ABB RAPID module: P36.mod

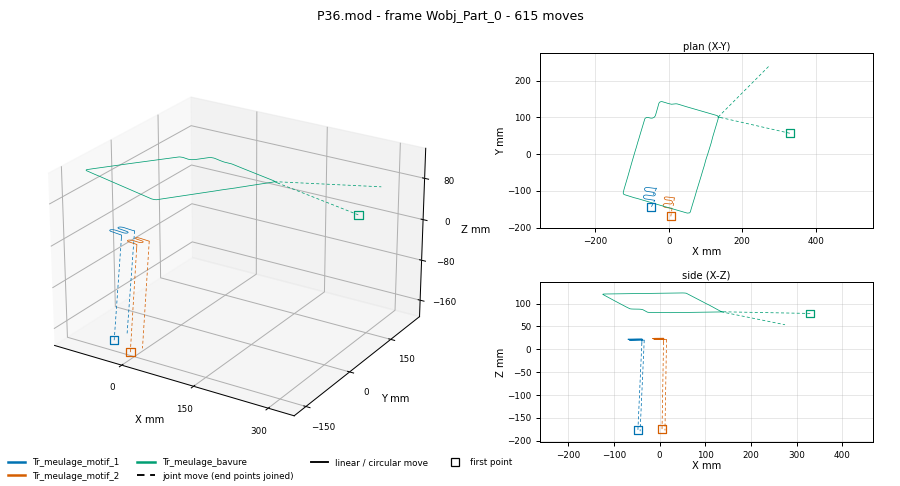
[picture p0: tool path of P36.mod in frame Wobj_Part_0, 615 of 623 moves have a stored position in this frame; points joined in program order, loops and branches not executed]
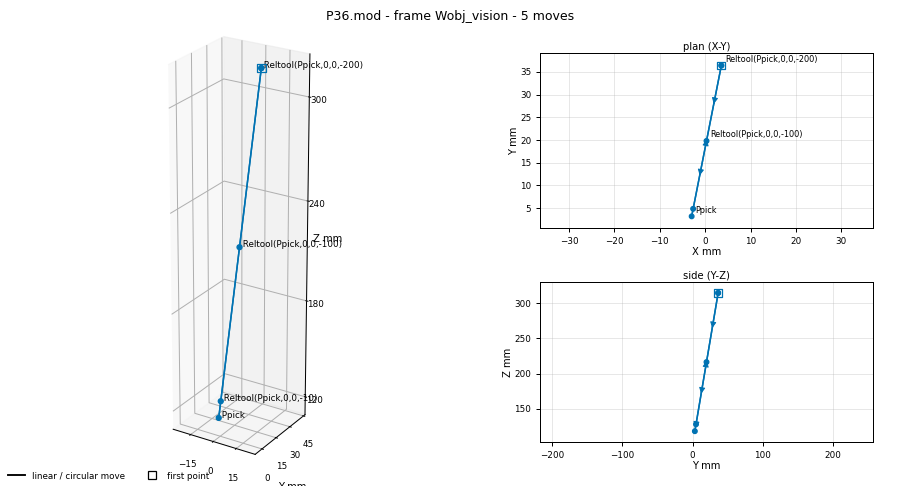
[picture p1: tool path of P36.mod in frame Wobj_vision, 5 of 623 moves have a stored position in this frame; points joined in program order, loops and branches not executed]
MODULE P36
	LOCAL CONST Speeddata vitesse_Tronconnage :=[10, 500, 0, 0];
	LOCAL CONST Robtarget Tr_meulage_motif_1_App1 :=[[-47.3344757449952,-143.415724704918,-176.118398279714],[-0.000994403231452177,0.0225685468013881,0.0440075228376034,0.998775755508305],[0,0,0,0],[8.999999E+09,8.999999E+09,8.999999E+09,8.999999E+09,8.999999E+09,8.999999E+09]];
	LOCAL CONST Robtarget Tr_meulage_motif_1_App2 :=[[-38.7855564044373,-126.704810844621,12.9521211992956],[-0.000994403231452177,0.0225685468013881,0.0440075228376034,0.998775755508305],[0,0,0,0],[8.999999E+09,8.999999E+09,8.999999E+09,8.999999E+09,8.999999E+09,8.999999E+09]];
	LOCAL CONST Robtarget Tr_meulage_motif_1_P0 :=[[-38.33561328125,-125.8252890625,22.903201171875],[-0.000994403231452177,0.0225685468013881,0.0440075228376034,0.998775755508305],[0,0,0,0],[8.999999E+09,8.999999E+09,8.999999E+09,8.999999E+09,8.999999E+09,8.999999E+09]];
	LOCAL CONST Robtarget Tr_meulage_motif_1_P1 :=[[-39.3248359375,-125.679359375,22.8911484375],[-0.000994403231452177,0.0225685468013881,0.0440075228376034,0.998775755508305],[0,0,0,0],[8.999999E+09,8.999999E+09,8.999999E+09,8.999999E+09,8.999999E+09,8.999999E+09]];
	LOCAL CONST Robtarget Tr_meulage_motif_1_P2 :=[[-40.3140546875,-125.533421875,22.879095703125],[-0.000994403231452177,0.0225685468013881,0.0440075228376034,0.998775755508305],[0,0,0,0],[8.999999E+09,8.999999E+09,8.999999E+09,8.999999E+09,8.999999E+09,8.999999E+09]];
	LOCAL CONST Robtarget Tr_meulage_motif_1_P3 :=[[-41.30327734375,-125.3874921875,22.867041015625],[-0.000994403231452177,0.0225685468013881,0.0440075228376034,0.998775755508305],[0,0,0,0],[8.999999E+09,8.999999E+09,8.999999E+09,8.999999E+09,8.999999E+09,8.999999E+09]];
	LOCAL CONST Robtarget Tr_meulage_motif_1_P4 :=[[-42.29249609375,-125.2415546875,22.85498828125],[-0.000994403231452177,0.0225685468013881,0.0440075228376034,0.998775755508305],[0,0,0,0],[8.999999E+09,8.999999E+09,8.999999E+09,8.999999E+09,8.999999E+09,8.999999E+09]];
	LOCAL CONST Robtarget Tr_meulage_motif_1_P5 :=[[-43.28171875,-125.095625,22.842935546875],[-0.000994403231452177,0.0225685468013881,0.0440075228376034,0.998775755508305],[0,0,0,0],[8.999999E+09,8.999999E+09,8.999999E+09,8.999999E+09,8.999999E+09,8.999999E+09]];
	LOCAL CONST Robtarget Tr_meulage_motif_1_P6 :=[[-44.2709375,-124.9496953125,22.8308828125],[-0.000994403231452177,0.0225685468013881,0.0440075228376034,0.998775755508305],[0,0,0,0],[8.999999E+09,8.999999E+09,8.999999E+09,8.999999E+09,8.999999E+09,8.999999E+09]];
	LOCAL CONST Robtarget Tr_meulage_motif_1_P7 :=[[-45.26016015625,-124.8037578125,22.818828125],[-0.000994403231452177,0.0225685468013881,0.0440075228376034,0.998775755508305],[0,0,0,0],[8.999999E+09,8.999999E+09,8.999999E+09,8.999999E+09,8.999999E+09,8.999999E+09]];
	LOCAL CONST Robtarget Tr_meulage_motif_1_P8 :=[[-46.2493828125,-124.657828125,22.806775390625],[-0.000994403231452177,0.0225685468013881,0.0440075228376034,0.998775755508305],[0,0,0,0],[8.999999E+09,8.999999E+09,8.999999E+09,8.999999E+09,8.999999E+09,8.999999E+09]];
	LOCAL CONST Robtarget Tr_meulage_motif_1_P9 :=[[-47.2386015625,-124.511890625,22.79472265625],[-0.000994403231452177,0.0225685468013881,0.0440075228376034,0.998775755508305],[0,0,0,0],[8.999999E+09,8.999999E+09,8.999999E+09,8.999999E+09,8.999999E+09,8.999999E+09]];
	LOCAL CONST Robtarget Tr_meulage_motif_1_P10 :=[[-48.22782421875,-124.3659609375,22.782669921875],[-0.000994403231452177,0.0225685468013881,0.0440075228376034,0.998775755508305],[0,0,0,0],[8.999999E+09,8.999999E+09,8.999999E+09,8.999999E+09,8.999999E+09,8.999999E+09]];
	LOCAL CONST Robtarget Tr_meulage_motif_1_P11 :=[[-49.21704296875,-124.2200234375,22.770615234375],[-0.000994403231452177,0.0225685468013881,0.0440075228376034,0.998775755508305],[0,0,0,0],[8.999999E+09,8.999999E+09,8.999999E+09,8.999999E+09,8.999999E+09,8.999999E+09]];
	LOCAL CONST Robtarget Tr_meulage_motif_1_P12 :=[[-50.206265625,-124.07409375,22.7585625],[-0.000994403231452177,0.0225685468013881,0.0440075228376034,0.998775755508305],[0,0,0,0],[8.999999E+09,8.999999E+09,8.999999E+09,8.999999E+09,8.999999E+09,8.999999E+09]];
	LOCAL CONST Robtarget Tr_meulage_motif_1_P13 :=[[-51.195484375,-123.92815625,22.746509765625],[-0.000994403231452177,0.0225685468013881,0.0440075228376034,0.998775755508305],[0,0,0,0],[8.999999E+09,8.999999E+09,8.999999E+09,8.999999E+09,8.999999E+09,8.999999E+09]];
	LOCAL CONST Robtarget Tr_meulage_motif_1_P14 :=[[-52.18470703125,-123.7822265625,22.734455078125],[-0.000994403231452177,0.0225685468013881,0.0440075228376034,0.998775755508305],[0,0,0,0],[8.999999E+09,8.999999E+09,8.999999E+09,8.999999E+09,8.999999E+09,8.999999E+09]];
	LOCAL CONST Robtarget Tr_meulage_motif_1_P15 :=[[-53.1739296875,-123.6362890625,22.72240234375],[-0.000994403231452177,0.0225685468013881,0.0440075228376034,0.998775755508305],[0,0,0,0],[8.999999E+09,8.999999E+09,8.999999E+09,8.999999E+09,8.999999E+09,8.999999E+09]];
	LOCAL CONST Robtarget Tr_meulage_motif_1_P16 :=[[-54.1631484375,-123.490359375,22.710349609375],[-0.000994403231452177,0.0225685468013881,0.0440075228376034,0.998775755508305],[0,0,0,0],[8.999999E+09,8.999999E+09,8.999999E+09,8.999999E+09,8.999999E+09,8.999999E+09]];
	LOCAL CONST Robtarget Tr_meulage_motif_1_P17 :=[[-55.15237109375,-123.344421875,22.698296875],[-0.000994403231452177,0.0225685468013881,0.0440075228376034,0.998775755508305],[0,0,0,0],[8.999999E+09,8.999999E+09,8.999999E+09,8.999999E+09,8.999999E+09,8.999999E+09]];
	LOCAL CONST Robtarget Tr_meulage_motif_1_P18 :=[[-56.14158984375,-123.1984921875,22.6862421875],[-0.000994403231452177,0.0225685468013881,0.0440075228376034,0.998775755508305],[0,0,0,0],[8.999999E+09,8.999999E+09,8.999999E+09,8.999999E+09,8.999999E+09,8.999999E+09]];
	LOCAL CONST Robtarget Tr_meulage_motif_1_P19 :=[[-57.1308125,-123.0525546875,22.674189453125],[-0.000994403231452177,0.0225685468013881,0.0440075228376034,0.998775755508305],[0,0,0,0],[8.999999E+09,8.999999E+09,8.999999E+09,8.999999E+09,8.999999E+09,8.999999E+09]];
	LOCAL CONST Robtarget Tr_meulage_motif_1_P20 :=[[-58.12003125,-122.906625,22.66213671875],[-0.000994403231452177,0.0225685468013881,0.0440075228376034,0.998775755508305],[0,0,0,0],[8.999999E+09,8.999999E+09,8.999999E+09,8.999999E+09,8.999999E+09,8.999999E+09]];
	LOCAL CONST Robtarget Tr_meulage_motif_1_P21 :=[[-59.10925390625,-122.7606875,22.650083984375],[-0.000994403231452177,0.0225685468013881,0.0440075228376034,0.998775755508305],[0,0,0,0],[8.999999E+09,8.999999E+09,8.999999E+09,8.999999E+09,8.999999E+09,8.999999E+09]];
	LOCAL CONST Robtarget Tr_meulage_motif_1_P22 :=[[-60.0984765625,-122.6147578125,22.638029296875],[-0.000994403231452177,0.0225685468013881,0.0440075228376034,0.998775755508305],[0,0,0,0],[8.999999E+09,8.999999E+09,8.999999E+09,8.999999E+09,8.999999E+09,8.999999E+09]];
	LOCAL CONST Robtarget Tr_meulage_motif_1_P23 :=[[-61.0876953125,-122.4688203125,22.6259765625],[-0.000994403231452177,0.0225685468013881,0.0440075228376034,0.998775755508305],[0,0,0,0],[8.999999E+09,8.999999E+09,8.999999E+09,8.999999E+09,8.999999E+09,8.999999E+09]];
	LOCAL CONST Robtarget Tr_meulage_motif_1_P24 :=[[-62.07691796875,-122.322890625,22.613923828125],[-0.000994403231452177,0.0225685468013881,0.0440075228376034,0.998775755508305],[0,0,0,0],[8.999999E+09,8.999999E+09,8.999999E+09,8.999999E+09,8.999999E+09,8.999999E+09]];
	LOCAL CONST Robtarget Tr_meulage_motif_1_P25 :=[[-63.06613671875,-122.176953125,22.601869140625],[-0.000994403231452177,0.0225685468013881,0.0440075228376034,0.998775755508305],[0,0,0,0],[8.999999E+09,8.999999E+09,8.999999E+09,8.999999E+09,8.999999E+09,8.999999E+09]];
	LOCAL CONST Robtarget Tr_meulage_motif_1_P26 :=[[-64.03180859375,-121.92315625,22.57997265625],[-0.000994403231452177,0.0225685468013881,0.0440075228376034,0.998775755508305],[0,0,0,0],[8.999999E+09,8.999999E+09,8.999999E+09,8.999999E+09,8.999999E+09,8.999999E+09]];
	LOCAL CONST Robtarget Tr_meulage_motif_1_P27 :=[[-64.93718359375,-121.576984375,22.54959765625],[-0.000994403231452177,0.0225685468013881,0.0440075228376034,0.998775755508305],[0,0,0,0],[8.999999E+09,8.999999E+09,8.999999E+09,8.999999E+09,8.999999E+09,8.999999E+09]];
	LOCAL CONST Robtarget Tr_meulage_motif_1_P28 :=[[-65.74090625,-121.1847421875,22.51490234375],[-0.000994403231452177,0.0225685468013881,0.0440075228376034,0.998775755508305],[0,0,0,0],[8.999999E+09,8.999999E+09,8.999999E+09,8.999999E+09,8.999999E+09,8.999999E+09]];
	LOCAL CONST Robtarget Tr_meulage_motif_1_P29 :=[[-66.4423515625,-120.8034609375,22.481080078125],[-0.000994403231452177,0.0225685468013881,0.0440075228376034,0.998775755508305],[0,0,0,0],[8.999999E+09,8.999999E+09,8.999999E+09,8.999999E+09,8.999999E+09,8.999999E+09]];
	LOCAL CONST Robtarget Tr_meulage_motif_1_P30 :=[[-67.4413359375,-120.0358125,22.412470703125],[-0.000994403231452177,0.0225685468013881,0.0440075228376034,0.998775755508305],[0,0,0,0],[8.999999E+09,8.999999E+09,8.999999E+09,8.999999E+09,8.999999E+09,8.999999E+09]];
	LOCAL CONST Robtarget Tr_meulage_motif_1_P31 :=[[-68.3300546875,-119.05134375,22.323998046875],[-0.000994403231452177,0.0225685468013881,0.0440075228376034,0.998775755508305],[0,0,0,0],[8.999999E+09,8.999999E+09,8.999999E+09,8.999999E+09,8.999999E+09,8.999999E+09]];
	LOCAL CONST Robtarget Tr_meulage_motif_1_P32 :=[[-69.0186484375,-117.918984375,22.2218203125],[-0.000994403231452177,0.0225685468013881,0.0440075228376034,0.998775755508305],[0,0,0,0],[8.999999E+09,8.999999E+09,8.999999E+09,8.999999E+09,8.999999E+09,8.999999E+09]];
	LOCAL CONST Robtarget Tr_meulage_motif_1_P33 :=[[-69.338109375,-116.7481484375,22.115685546875],[-0.000994403231452177,0.0225685468013881,0.0440075228376034,0.998775755508305],[0,0,0,0],[8.999999E+09,8.999999E+09,8.999999E+09,8.999999E+09,8.999999E+09,8.999999E+09]];
	LOCAL CONST Robtarget Tr_meulage_motif_1_P34 :=[[-69.26296875,-116.058578125,22.0528515625],[-0.000994403231452177,0.0225685468013881,0.0440075228376034,0.998775755508305],[0,0,0,0],[8.999999E+09,8.999999E+09,8.999999E+09,8.999999E+09,8.999999E+09,8.999999E+09]];
	LOCAL CONST Robtarget Tr_meulage_motif_1_P35 :=[[-69.1661484375,-115.40715625,21.9934609375],[-0.000994403231452177,0.0225685468013881,0.0440075228376034,0.998775755508305],[0,0,0,0],[8.999999E+09,8.999999E+09,8.999999E+09,8.999999E+09,8.999999E+09,8.999999E+09]];
	LOCAL CONST Robtarget Tr_meulage_motif_1_P36 :=[[-69.0150625,-114.7638984375,21.93474609375],[-0.000994403231452177,0.0225685468013881,0.0440075228376034,0.998775755508305],[0,0,0,0],[8.999999E+09,8.999999E+09,8.999999E+09,8.999999E+09,8.999999E+09,8.999999E+09]];
	LOCAL CONST Robtarget Tr_meulage_motif_1_P37 :=[[-68.360890625,-113.7512265625,21.841796875],[-0.000994403231452177,0.0225685468013881,0.0440075228376034,0.998775755508305],[0,0,0,0],[8.999999E+09,8.999999E+09,8.999999E+09,8.999999E+09,8.999999E+09,8.999999E+09]];
	LOCAL CONST Robtarget Tr_meulage_motif_1_P38 :=[[-67.3661015625,-112.884578125,21.7617109375],[-0.000994403231452177,0.0225685468013881,0.0440075228376034,0.998775755508305],[0,0,0,0],[8.999999E+09,8.999999E+09,8.999999E+09,8.999999E+09,8.999999E+09,8.999999E+09]];
	LOCAL CONST Robtarget Tr_meulage_motif_1_P39 :=[[-66.232359375,-112.217375,21.6996015625],[-0.000994403231452177,0.0225685468013881,0.0440075228376034,0.998775755508305],[0,0,0,0],[8.999999E+09,8.999999E+09,8.999999E+09,8.999999E+09,8.999999E+09,8.999999E+09]];
	LOCAL CONST Robtarget Tr_meulage_motif_1_P40 :=[[-65.4947265625,-111.9277734375,21.672337890625],[-0.000994403231452177,0.0225685468013881,0.0440075228376034,0.998775755508305],[0,0,0,0],[8.999999E+09,8.999999E+09,8.999999E+09,8.999999E+09,8.999999E+09,8.999999E+09]];
	LOCAL CONST Robtarget Tr_meulage_motif_1_P41 :=[[-64.27766796875,-111.6165,21.642509765625],[-0.000994403231452177,0.0225685468013881,0.0440075228376034,0.998775755508305],[0,0,0,0],[8.999999E+09,8.999999E+09,8.999999E+09,8.999999E+09,8.999999E+09,8.999999E+09]];
	LOCAL CONST Robtarget Tr_meulage_motif_1_P42 :=[[-63.40307421875,-111.47965625,21.628974609375],[-0.000994403231452177,0.0225685468013881,0.0440075228376034,0.998775755508305],[0,0,0,0],[8.999999E+09,8.999999E+09,8.999999E+09,8.999999E+09,8.999999E+09,8.999999E+09]];
	LOCAL CONST Robtarget Tr_meulage_motif_1_P43 :=[[-62.4511796875,-111.414234375,21.62184375],[-0.000994403231452177,0.0225685468013881,0.0440075228376034,0.998775755508305],[0,0,0,0],[8.999999E+09,8.999999E+09,8.999999E+09,8.999999E+09,8.999999E+09,8.999999E+09]];
	LOCAL CONST Robtarget Tr_meulage_motif_1_P44 :=[[-61.464296875,-111.4505,21.623921875],[-0.000994403231452177,0.0225685468013881,0.0440075228376034,0.998775755508305],[0,0,0,0],[8.999999E+09,8.999999E+09,8.999999E+09,8.999999E+09,8.999999E+09,8.999999E+09]];
	LOCAL CONST Robtarget Tr_meulage_motif_1_P45 :=[[-60.4662421875,-111.486390625,21.625953125],[-0.000994403231452177,0.0225685468013881,0.0440075228376034,0.998775755508305],[0,0,0,0],[8.999999E+09,8.999999E+09,8.999999E+09,8.999999E+09,8.999999E+09,8.999999E+09]];
	LOCAL CONST Robtarget Tr_meulage_motif_1_P46 :=[[-59.47701953125,-111.632328125,21.638005859375],[-0.000994403231452177,0.0225685468013881,0.0440075228376034,0.998775755508305],[0,0,0,0],[8.999999E+09,8.999999E+09,8.999999E+09,8.999999E+09,8.999999E+09,8.999999E+09]];
	LOCAL CONST Robtarget Tr_meulage_motif_1_P47 :=[[-58.487796875,-111.7782578125,21.65005859375],[-0.000994403231452177,0.0225685468013881,0.0440075228376034,0.998775755508305],[0,0,0,0],[8.999999E+09,8.999999E+09,8.999999E+09,8.999999E+09,8.999999E+09,8.999999E+09]];
	LOCAL CONST Robtarget Tr_meulage_motif_1_P48 :=[[-57.498578125,-111.9241953125,21.66211328125],[-0.000994403231452177,0.0225685468013881,0.0440075228376034,0.998775755508305],[0,0,0,0],[8.999999E+09,8.999999E+09,8.999999E+09,8.999999E+09,8.999999E+09,8.999999E+09]];
	LOCAL CONST Robtarget Tr_meulage_motif_1_P49 :=[[-56.50935546875,-112.070125,21.674166015625],[-0.000994403231452177,0.0225685468013881,0.0440075228376034,0.998775755508305],[0,0,0,0],[8.999999E+09,8.999999E+09,8.999999E+09,8.999999E+09,8.999999E+09,8.999999E+09]];
	LOCAL CONST Robtarget Tr_meulage_motif_1_P50 :=[[-55.52013671875,-112.2160625,21.68621875],[-0.000994403231452177,0.0225685468013881,0.0440075228376034,0.998775755508305],[0,0,0,0],[8.999999E+09,8.999999E+09,8.999999E+09,8.999999E+09,8.999999E+09,8.999999E+09]];
	LOCAL CONST Robtarget Tr_meulage_motif_1_P51 :=[[-54.5309140625,-112.3619921875,21.698271484375],[-0.000994403231452177,0.0225685468013881,0.0440075228376034,0.998775755508305],[0,0,0,0],[8.999999E+09,8.999999E+09,8.999999E+09,8.999999E+09,8.999999E+09,8.999999E+09]];
	LOCAL CONST Robtarget Tr_meulage_motif_1_P52 :=[[-53.5416953125,-112.5079296875,21.710326171875],[-0.000994403231452177,0.0225685468013881,0.0440075228376034,0.998775755508305],[0,0,0,0],[8.999999E+09,8.999999E+09,8.999999E+09,8.999999E+09,8.999999E+09,8.999999E+09]];
	LOCAL CONST Robtarget Tr_meulage_motif_1_P53 :=[[-52.55247265625,-112.653859375,21.72237890625],[-0.000994403231452177,0.0225685468013881,0.0440075228376034,0.998775755508305],[0,0,0,0],[8.999999E+09,8.999999E+09,8.999999E+09,8.999999E+09,8.999999E+09,8.999999E+09]];
	LOCAL CONST Robtarget Tr_meulage_motif_1_P54 :=[[-51.56325,-112.799796875,21.734431640625],[-0.000994403231452177,0.0225685468013881,0.0440075228376034,0.998775755508305],[0,0,0,0],[8.999999E+09,8.999999E+09,8.999999E+09,8.999999E+09,8.999999E+09,8.999999E+09]];
	LOCAL CONST Robtarget Tr_meulage_motif_1_P55 :=[[-50.57403125,-112.9457265625,21.746486328125],[-0.000994403231452177,0.0225685468013881,0.0440075228376034,0.998775755508305],[0,0,0,0],[8.999999E+09,8.999999E+09,8.999999E+09,8.999999E+09,8.999999E+09,8.999999E+09]];
	LOCAL CONST Robtarget Tr_meulage_motif_1_P56 :=[[-49.58480859375,-113.0916640625,21.7585390625],[-0.000994403231452177,0.0225685468013881,0.0440075228376034,0.998775755508305],[0,0,0,0],[8.999999E+09,8.999999E+09,8.999999E+09,8.999999E+09,8.999999E+09,8.999999E+09]];
	LOCAL CONST Robtarget Tr_meulage_motif_1_P57 :=[[-48.59558984375,-113.23759375,21.770591796875],[-0.000994403231452177,0.0225685468013881,0.0440075228376034,0.998775755508305],[0,0,0,0],[8.999999E+09,8.999999E+09,8.999999E+09,8.999999E+09,8.999999E+09,8.999999E+09]];
	LOCAL CONST Robtarget Tr_meulage_motif_1_P58 :=[[-47.6063671875,-113.38353125,21.78264453125],[-0.000994403231452177,0.0225685468013881,0.0440075228376034,0.998775755508305],[0,0,0,0],[8.999999E+09,8.999999E+09,8.999999E+09,8.999999E+09,8.999999E+09,8.999999E+09]];
	LOCAL CONST Robtarget Tr_meulage_motif_1_P59 :=[[-46.6171484375,-113.5294609375,21.79469921875],[-0.000994403231452177,0.0225685468013881,0.0440075228376034,0.998775755508305],[0,0,0,0],[8.999999E+09,8.999999E+09,8.999999E+09,8.999999E+09,8.999999E+09,8.999999E+09]];
	LOCAL CONST Robtarget Tr_meulage_motif_1_P60 :=[[-45.62792578125,-113.6753984375,21.806751953125],[-0.000994403231452177,0.0225685468013881,0.0440075228376034,0.998775755508305],[0,0,0,0],[8.999999E+09,8.999999E+09,8.999999E+09,8.999999E+09,8.999999E+09,8.999999E+09]];
	LOCAL CONST Robtarget Tr_meulage_motif_1_P61 :=[[-44.638703125,-113.821328125,21.8188046875],[-0.000994403231452177,0.0225685468013881,0.0440075228376034,0.998775755508305],[0,0,0,0],[8.999999E+09,8.999999E+09,8.999999E+09,8.999999E+09,8.999999E+09,8.999999E+09]];
	LOCAL CONST Robtarget Tr_meulage_motif_1_P62 :=[[-43.649484375,-113.967265625,21.830857421875],[-0.000994403231452177,0.0225685468013881,0.0440075228376034,0.998775755508305],[0,0,0,0],[8.999999E+09,8.999999E+09,8.999999E+09,8.999999E+09,8.999999E+09,8.999999E+09]];
	LOCAL CONST Robtarget Tr_meulage_motif_1_P63 :=[[-42.65142578125,-114.0031640625,21.832888671875],[-0.000994403231452177,0.0225685468013881,0.0440075228376034,0.998775755508305],[0,0,0,0],[8.999999E+09,8.999999E+09,8.999999E+09,8.999999E+09,8.999999E+09,8.999999E+09]];
	LOCAL CONST Robtarget Tr_meulage_motif_1_P64 :=[[-41.68420703125,-113.9332421875,21.825330078125],[-0.000994403231452177,0.0225685468013881,0.0440075228376034,0.998775755508305],[0,0,0,0],[8.999999E+09,8.999999E+09,8.999999E+09,8.999999E+09,8.999999E+09,8.999999E+09]];
	LOCAL CONST Robtarget Tr_meulage_motif_1_P65 :=[[-40.800875,-113.789875,21.81119140625],[-0.000994403231452177,0.0225685468013881,0.0440075228376034,0.998775755508305],[0,0,0,0],[8.999999E+09,8.999999E+09,8.999999E+09,8.999999E+09,8.999999E+09,8.999999E+09]];
	LOCAL CONST Robtarget Tr_meulage_motif_1_P66 :=[[-40.0525078125,-113.5940703125,21.79244921875],[-0.000994403231452177,0.0225685468013881,0.0440075228376034,0.998775755508305],[0,0,0,0],[8.999999E+09,8.999999E+09,8.999999E+09,8.999999E+09,8.999999E+09,8.999999E+09]];
	LOCAL CONST Robtarget Tr_meulage_motif_1_P67 :=[[-38.93217578125,-113.0923515625,21.745412109375],[-0.000994403231452177,0.0225685468013881,0.0440075228376034,0.998775755508305],[0,0,0,0],[8.999999E+09,8.999999E+09,8.999999E+09,8.999999E+09,8.999999E+09,8.999999E+09]];
	LOCAL CONST Robtarget Tr_meulage_motif_1_P68 :=[[-37.90789453125,-112.3354453125,21.675275390625],[-0.000994403231452177,0.0225685468013881,0.0440075228376034,0.998775755508305],[0,0,0,0],[8.999999E+09,8.999999E+09,8.999999E+09,8.999999E+09,8.999999E+09,8.999999E+09]];
	LOCAL CONST Robtarget Tr_meulage_motif_1_P69 :=[[-37.22552734375,-111.38303125,21.5877734375],[-0.000994403231452177,0.0225685468013881,0.0440075228376034,0.998775755508305],[0,0,0,0],[8.999999E+09,8.999999E+09,8.999999E+09,8.999999E+09,8.999999E+09,8.999999E+09]];
	LOCAL CONST Robtarget Tr_meulage_motif_1_P70 :=[[-36.941234375,-110.727078125,21.527740234375],[-0.000994403231452177,0.0225685468013881,0.0440075228376034,0.998775755508305],[0,0,0,0],[8.999999E+09,8.999999E+09,8.999999E+09,8.999999E+09,8.999999E+09,8.999999E+09]];
	LOCAL CONST Robtarget Tr_meulage_motif_1_P71 :=[[-36.76533203125,-109.97784375,21.4593515625],[-0.000994403231452177,0.0225685468013881,0.0440075228376034,0.998775755508305],[0,0,0,0],[8.999999E+09,8.999999E+09,8.999999E+09,8.999999E+09,8.999999E+09,8.999999E+09]];
	LOCAL CONST Robtarget Tr_meulage_motif_1_P72 :=[[-36.71881640625,-109.209640625,21.3893984375],[-0.000994403231452177,0.0225685468013881,0.0440075228376034,0.998775755508305],[0,0,0,0],[8.999999E+09,8.999999E+09,8.999999E+09,8.999999E+09,8.999999E+09,8.999999E+09]];
	LOCAL CONST Robtarget Tr_meulage_motif_1_P73 :=[[-36.97161328125,-108.0566328125,21.284802734375],[-0.000994403231452177,0.0225685468013881,0.0440075228376034,0.998775755508305],[0,0,0,0],[8.999999E+09,8.999999E+09,8.999999E+09,8.999999E+09,8.999999E+09,8.999999E+09]];
	LOCAL CONST Robtarget Tr_meulage_motif_1_P74 :=[[-37.29569921875,-107.4191875,21.227205078125],[-0.000994403231452177,0.0225685468013881,0.0440075228376034,0.998775755508305],[0,0,0,0],[8.999999E+09,8.999999E+09,8.999999E+09,8.999999E+09,8.999999E+09,8.999999E+09]];
	LOCAL CONST Robtarget Tr_meulage_motif_1_P75 :=[[-38.0433671875,-106.4157890625,21.136833984375],[-0.000994403231452177,0.0225685468013881,0.0440075228376034,0.998775755508305],[0,0,0,0],[8.999999E+09,8.999999E+09,8.999999E+09,8.999999E+09,8.999999E+09,8.999999E+09]];
	LOCAL CONST Robtarget Tr_meulage_motif_1_P76 :=[[-38.56207421875,-105.9221640625,21.0925625],[-0.000994403231452177,0.0225685468013881,0.0440075228376034,0.998775755508305],[0,0,0,0],[8.999999E+09,8.999999E+09,8.999999E+09,8.999999E+09,8.999999E+09,8.999999E+09]];
	LOCAL CONST Robtarget Tr_meulage_motif_1_P77 :=[[-39.58826171875,-105.223015625,21.030220703125],[-0.000994403231452177,0.0225685468013881,0.0440075228376034,0.998775755508305],[0,0,0,0],[8.999999E+09,8.999999E+09,8.999999E+09,8.999999E+09,8.999999E+09,8.999999E+09]];
	LOCAL CONST Robtarget Tr_meulage_motif_1_P78 :=[[-40.3616875,-104.8114296875,20.993728515625],[-0.000994403231452177,0.0225685468013881,0.0440075228376034,0.998775755508305],[0,0,0,0],[8.999999E+09,8.999999E+09,8.999999E+09,8.999999E+09,8.999999E+09,8.999999E+09]];
	LOCAL CONST Robtarget Tr_meulage_motif_1_P79 :=[[-41.253703125,-104.4739921875,20.964130859375],[-0.000994403231452177,0.0225685468013881,0.0440075228376034,0.998775755508305],[0,0,0,0],[8.999999E+09,8.999999E+09,8.999999E+09,8.999999E+09,8.999999E+09,8.999999E+09]];
	LOCAL CONST Robtarget Tr_meulage_motif_1_P80 :=[[-42.20878515625,-104.223765625,20.942546875],[-0.000994403231452177,0.0225685468013881,0.0440075228376034,0.998775755508305],[0,0,0,0],[8.999999E+09,8.999999E+09,8.999999E+09,8.999999E+09,8.999999E+09,8.999999E+09]];
	LOCAL CONST Robtarget Tr_meulage_motif_1_P81 :=[[-43.174453125,-103.96996875,20.920650390625],[-0.000994403231452177,0.0225685468013881,0.0440075228376034,0.998775755508305],[0,0,0,0],[8.999999E+09,8.999999E+09,8.999999E+09,8.999999E+09,8.999999E+09,8.999999E+09]];
	LOCAL CONST Robtarget Tr_meulage_motif_1_P82 :=[[-44.16367578125,-103.8240390625,20.90859765625],[-0.000994403231452177,0.0225685468013881,0.0440075228376034,0.998775755508305],[0,0,0,0],[8.999999E+09,8.999999E+09,8.999999E+09,8.999999E+09,8.999999E+09,8.999999E+09]];
	LOCAL CONST Robtarget Tr_meulage_motif_1_P83 :=[[-45.15289453125,-103.6781015625,20.89654296875],[-0.000994403231452177,0.0225685468013881,0.0440075228376034,0.998775755508305],[0,0,0,0],[8.999999E+09,8.999999E+09,8.999999E+09,8.999999E+09,8.999999E+09,8.999999E+09]];
	LOCAL CONST Robtarget Tr_meulage_motif_1_P84 :=[[-46.1421171875,-103.532171875,20.884490234375],[-0.000994403231452177,0.0225685468013881,0.0440075228376034,0.998775755508305],[0,0,0,0],[8.999999E+09,8.999999E+09,8.999999E+09,8.999999E+09,8.999999E+09,8.999999E+09]];
	LOCAL CONST Robtarget Tr_meulage_motif_1_P85 :=[[-47.1313359375,-103.386234375,20.8724375],[-0.000994403231452177,0.0225685468013881,0.0440075228376034,0.998775755508305],[0,0,0,0],[8.999999E+09,8.999999E+09,8.999999E+09,8.999999E+09,8.999999E+09,8.999999E+09]];
	LOCAL CONST Robtarget Tr_meulage_motif_1_P86 :=[[-48.12055859375,-103.2403046875,20.8603828125],[-0.000994403231452177,0.0225685468013881,0.0440075228376034,0.998775755508305],[0,0,0,0],[8.999999E+09,8.999999E+09,8.999999E+09,8.999999E+09,8.999999E+09,8.999999E+09]];
	LOCAL CONST Robtarget Tr_meulage_motif_1_P87 :=[[-49.10977734375,-103.0943671875,20.848330078125],[-0.000994403231452177,0.0225685468013881,0.0440075228376034,0.998775755508305],[0,0,0,0],[8.999999E+09,8.999999E+09,8.999999E+09,8.999999E+09,8.999999E+09,8.999999E+09]];
	LOCAL CONST Robtarget Tr_meulage_motif_1_P88 :=[[-50.099,-102.9484375,20.83627734375],[-0.000994403231452177,0.0225685468013881,0.0440075228376034,0.998775755508305],[0,0,0,0],[8.999999E+09,8.999999E+09,8.999999E+09,8.999999E+09,8.999999E+09,8.999999E+09]];
	LOCAL CONST Robtarget Tr_meulage_motif_1_P89 :=[[-51.08822265625,-102.8025,20.824224609375],[-0.000994403231452177,0.0225685468013881,0.0440075228376034,0.998775755508305],[0,0,0,0],[8.999999E+09,8.999999E+09,8.999999E+09,8.999999E+09,8.999999E+09,8.999999E+09]];
	LOCAL CONST Robtarget Tr_meulage_motif_1_P90 :=[[-52.07744140625,-102.6565703125,20.812169921875],[-0.000994403231452177,0.0225685468013881,0.0440075228376034,0.998775755508305],[0,0,0,0],[8.999999E+09,8.999999E+09,8.999999E+09,8.999999E+09,8.999999E+09,8.999999E+09]];
	LOCAL CONST Robtarget Tr_meulage_motif_1_P91 :=[[-53.0666640625,-102.5106328125,20.8001171875],[-0.000994403231452177,0.0225685468013881,0.0440075228376034,0.998775755508305],[0,0,0,0],[8.999999E+09,8.999999E+09,8.999999E+09,8.999999E+09,8.999999E+09,8.999999E+09]];
	LOCAL CONST Robtarget Tr_meulage_motif_1_P92 :=[[-54.0558828125,-102.364703125,20.788064453125],[-0.000994403231452177,0.0225685468013881,0.0440075228376034,0.998775755508305],[0,0,0,0],[8.999999E+09,8.999999E+09,8.999999E+09,8.999999E+09,8.999999E+09,8.999999E+09]];
	LOCAL CONST Robtarget Tr_meulage_motif_1_P93 :=[[-55.04510546875,-102.218765625,20.77601171875],[-0.000994403231452177,0.0225685468013881,0.0440075228376034,0.998775755508305],[0,0,0,0],[8.999999E+09,8.999999E+09,8.999999E+09,8.999999E+09,8.999999E+09,8.999999E+09]];
	LOCAL CONST Robtarget Tr_meulage_motif_1_P94 :=[[-56.03432421875,-102.0728359375,20.76395703125],[-0.000994403231452177,0.0225685468013881,0.0440075228376034,0.998775755508305],[0,0,0,0],[8.999999E+09,8.999999E+09,8.999999E+09,8.999999E+09,8.999999E+09,8.999999E+09]];
	LOCAL CONST Robtarget Tr_meulage_motif_1_P95 :=[[-57.023546875,-101.9268984375,20.751904296875],[-0.000994403231452177,0.0225685468013881,0.0440075228376034,0.998775755508305],[0,0,0,0],[8.999999E+09,8.999999E+09,8.999999E+09,8.999999E+09,8.999999E+09,8.999999E+09]];
	LOCAL CONST Robtarget Tr_meulage_motif_1_P96 :=[[-58.01276953125,-101.78096875,20.7398515625],[-0.000994403231452177,0.0225685468013881,0.0440075228376034,0.998775755508305],[0,0,0,0],[8.999999E+09,8.999999E+09,8.999999E+09,8.999999E+09,8.999999E+09,8.999999E+09]];
	LOCAL CONST Robtarget Tr_meulage_motif_1_P97 :=[[-59.00198828125,-101.63503125,20.727796875],[-0.000994403231452177,0.0225685468013881,0.0440075228376034,0.998775755508305],[0,0,0,0],[8.999999E+09,8.999999E+09,8.999999E+09,8.999999E+09,8.999999E+09,8.999999E+09]];
	LOCAL CONST Robtarget Tr_meulage_motif_1_P98 :=[[-59.9912109375,-101.4891015625,20.715744140625],[-0.000994403231452177,0.0225685468013881,0.0440075228376034,0.998775755508305],[0,0,0,0],[8.999999E+09,8.999999E+09,8.999999E+09,8.999999E+09,8.999999E+09,8.999999E+09]];
	LOCAL CONST Robtarget Tr_meulage_motif_1_P99 :=[[-60.95687890625,-101.2353046875,20.69384765625],[-0.000994403231452177,0.0225685468013881,0.0440075228376034,0.998775755508305],[0,0,0,0],[8.999999E+09,8.999999E+09,8.999999E+09,8.999999E+09,8.999999E+09,8.999999E+09]];
	LOCAL CONST Robtarget Tr_meulage_motif_1_P100 :=[[-61.86225390625,-100.8891328125,20.663470703125],[-0.000994403231452177,0.0225685468013881,0.0440075228376034,0.998775755508305],[0,0,0,0],[8.999999E+09,8.999999E+09,8.999999E+09,8.999999E+09,8.999999E+09,8.999999E+09]];
	LOCAL CONST Robtarget Tr_meulage_motif_1_P101 :=[[-62.6659765625,-100.4968828125,20.62877734375],[-0.000994403231452177,0.0225685468013881,0.0440075228376034,0.998775755508305],[0,0,0,0],[8.999999E+09,8.999999E+09,8.999999E+09,8.999999E+09,8.999999E+09,8.999999E+09]];
	LOCAL CONST Robtarget Tr_meulage_motif_1_P102 :=[[-63.36742578125,-100.115609375,20.594955078125],[-0.000994403231452177,0.0225685468013881,0.0440075228376034,0.998775755508305],[0,0,0,0],[8.999999E+09,8.999999E+09,8.999999E+09,8.999999E+09,8.999999E+09,8.999999E+09]];
	LOCAL CONST Robtarget Tr_meulage_motif_1_P103 :=[[-64.36640625,-99.3479609375,20.526345703125],[-0.000994403231452177,0.0225685468013881,0.0440075228376034,0.998775755508305],[0,0,0,0],[8.999999E+09,8.999999E+09,8.999999E+09,8.999999E+09,8.999999E+09,8.999999E+09]];
	LOCAL CONST Robtarget Tr_meulage_motif_1_P104 :=[[-65.255125,-98.363484375,20.437873046875],[-0.000994403231452177,0.0225685468013881,0.0440075228376034,0.998775755508305],[0,0,0,0],[8.999999E+09,8.999999E+09,8.999999E+09,8.999999E+09,8.999999E+09,8.999999E+09]];
	LOCAL CONST Robtarget Tr_meulage_motif_1_P105 :=[[-65.9437265625,-97.231125,20.3356953125],[-0.000994403231452177,0.0225685468013881,0.0440075228376034,0.998775755508305],[0,0,0,0],[8.999999E+09,8.999999E+09,8.999999E+09,8.999999E+09,8.999999E+09,8.999999E+09]];
	LOCAL CONST Robtarget Tr_meulage_motif_1_P106 :=[[-66.2631796875,-96.060296875,20.229560546875],[-0.000994403231452177,0.0225685468013881,0.0440075228376034,0.998775755508305],[0,0,0,0],[8.999999E+09,8.999999E+09,8.999999E+09,8.999999E+09,8.999999E+09,8.999999E+09]];
	LOCAL CONST Robtarget Tr_meulage_motif_1_P107 :=[[-66.188046875,-95.37071875,20.166724609375],[-0.000994403231452177,0.0225685468013881,0.0440075228376034,0.998775755508305],[0,0,0,0],[8.999999E+09,8.999999E+09,8.999999E+09,8.999999E+09,8.999999E+09,8.999999E+09]];
	LOCAL CONST Robtarget Tr_meulage_motif_1_P108 :=[[-66.09121875,-94.719296875,20.1073359375],[-0.000994403231452177,0.0225685468013881,0.0440075228376034,0.998775755508305],[0,0,0,0],[8.999999E+09,8.999999E+09,8.999999E+09,8.999999E+09,8.999999E+09,8.999999E+09]];
	LOCAL CONST Robtarget Tr_meulage_motif_1_P109 :=[[-65.9401328125,-94.0760390625,20.048619140625],[-0.000994403231452177,0.0225685468013881,0.0440075228376034,0.998775755508305],[0,0,0,0],[8.999999E+09,8.999999E+09,8.999999E+09,8.999999E+09,8.999999E+09,8.999999E+09]];
	LOCAL CONST Robtarget Tr_meulage_motif_1_P110 :=[[-65.28596484375,-93.063375,19.955671875],[-0.000994403231452177,0.0225685468013881,0.0440075228376034,0.998775755508305],[0,0,0,0],[8.999999E+09,8.999999E+09,8.999999E+09,8.999999E+09,8.999999E+09,8.999999E+09]];
	LOCAL CONST Robtarget Tr_meulage_motif_1_P111 :=[[-64.29117578125,-92.19671875,19.8755859375],[-0.000994403231452177,0.0225685468013881,0.0440075228376034,0.998775755508305],[0,0,0,0],[8.999999E+09,8.999999E+09,8.999999E+09,8.999999E+09,8.999999E+09,8.999999E+09]];
	LOCAL CONST Robtarget Tr_meulage_motif_1_P112 :=[[-63.15743359375,-91.529515625,19.813474609375],[-0.000994403231452177,0.0225685468013881,0.0440075228376034,0.998775755508305],[0,0,0,0],[8.999999E+09,8.999999E+09,8.999999E+09,8.999999E+09,8.999999E+09,8.999999E+09]];
	LOCAL CONST Robtarget Tr_meulage_motif_1_P113 :=[[-62.419796875,-91.239921875,19.786212890625],[-0.000994403231452177,0.0225685468013881,0.0440075228376034,0.998775755508305],[0,0,0,0],[8.999999E+09,8.999999E+09,8.999999E+09,8.999999E+09,8.999999E+09,8.999999E+09]];
	LOCAL CONST Robtarget Tr_meulage_motif_1_P114 :=[[-61.20273828125,-90.9286484375,19.756384765625],[-0.000994403231452177,0.0225685468013881,0.0440075228376034,0.998775755508305],[0,0,0,0],[8.999999E+09,8.999999E+09,8.999999E+09,8.999999E+09,8.999999E+09,8.999999E+09]];
	LOCAL CONST Robtarget Tr_meulage_motif_1_P115 :=[[-60.32814453125,-90.791796875,19.742849609375],[-0.000994403231452177,0.0225685468013881,0.0440075228376034,0.998775755508305],[0,0,0,0],[8.999999E+09,8.999999E+09,8.999999E+09,8.999999E+09,8.999999E+09,8.999999E+09]];
	LOCAL CONST Robtarget Tr_meulage_motif_1_P116 :=[[-59.37625390625,-90.726375,19.73571875],[-0.000994403231452177,0.0225685468013881,0.0440075228376034,0.998775755508305],[0,0,0,0],[8.999999E+09,8.999999E+09,8.999999E+09,8.999999E+09,8.999999E+09,8.999999E+09]];
	LOCAL CONST Robtarget Tr_meulage_motif_1_P117 :=[[-58.38937109375,-90.762640625,19.737796875],[-0.000994403231452177,0.0225685468013881,0.0440075228376034,0.998775755508305],[0,0,0,0],[8.999999E+09,8.999999E+09,8.999999E+09,8.999999E+09,8.999999E+09,8.999999E+09]];
	LOCAL CONST Robtarget Tr_meulage_motif_1_P118 :=[[-57.3913125,-90.7985390625,19.739826171875],[-0.000994403231452177,0.0225685468013881,0.0440075228376034,0.998775755508305],[0,0,0,0],[8.999999E+09,8.999999E+09,8.999999E+09,8.999999E+09,8.999999E+09,8.999999E+09]];
	LOCAL CONST Robtarget Tr_meulage_motif_1_P119 :=[[-56.40208984375,-90.9444765625,19.751880859375],[-0.000994403231452177,0.0225685468013881,0.0440075228376034,0.998775755508305],[0,0,0,0],[8.999999E+09,8.999999E+09,8.999999E+09,8.999999E+09,8.999999E+09,8.999999E+09]];
	LOCAL CONST Robtarget Tr_meulage_motif_1_P120 :=[[-55.41287109375,-91.09040625,19.76393359375],[-0.000994403231452177,0.0225685468013881,0.0440075228376034,0.998775755508305],[0,0,0,0],[8.999999E+09,8.999999E+09,8.999999E+09,8.999999E+09,8.999999E+09,8.999999E+09]];
	LOCAL CONST Robtarget Tr_meulage_motif_1_P121 :=[[-54.4236484375,-91.2363359375,19.775986328125],[-0.000994403231452177,0.0225685468013881,0.0440075228376034,0.998775755508305],[0,0,0,0],[8.999999E+09,8.999999E+09,8.999999E+09,8.999999E+09,8.999999E+09,8.999999E+09]];
	LOCAL CONST Robtarget Tr_meulage_motif_1_P122 :=[[-53.4344296875,-91.3822734375,19.788041015625],[-0.000994403231452177,0.0225685468013881,0.0440075228376034,0.998775755508305],[0,0,0,0],[8.999999E+09,8.999999E+09,8.999999E+09,8.999999E+09,8.999999E+09,8.999999E+09]];
	LOCAL CONST Robtarget Tr_meulage_motif_1_P123 :=[[-52.44520703125,-91.528203125,19.80009375],[-0.000994403231452177,0.0225685468013881,0.0440075228376034,0.998775755508305],[0,0,0,0],[8.999999E+09,8.999999E+09,8.999999E+09,8.999999E+09,8.999999E+09,8.999999E+09]];
	LOCAL CONST Robtarget Tr_meulage_motif_1_P124 :=[[-51.45598828125,-91.674140625,19.812146484375],[-0.000994403231452177,0.0225685468013881,0.0440075228376034,0.998775755508305],[0,0,0,0],[8.999999E+09,8.999999E+09,8.999999E+09,8.999999E+09,8.999999E+09,8.999999E+09]];
	LOCAL CONST Robtarget Tr_meulage_motif_1_P125 :=[[-50.466765625,-91.8200703125,19.82419921875],[-0.000994403231452177,0.0225685468013881,0.0440075228376034,0.998775755508305],[0,0,0,0],[8.999999E+09,8.999999E+09,8.999999E+09,8.999999E+09,8.999999E+09,8.999999E+09]];
	LOCAL CONST Robtarget Tr_meulage_motif_1_P126 :=[[-49.47754296875,-91.9660078125,19.83625390625],[-0.000994403231452177,0.0225685468013881,0.0440075228376034,0.998775755508305],[0,0,0,0],[8.999999E+09,8.999999E+09,8.999999E+09,8.999999E+09,8.999999E+09,8.999999E+09]];
	LOCAL CONST Robtarget Tr_meulage_motif_1_P127 :=[[-48.48832421875,-92.1119375,19.848306640625],[-0.000994403231452177,0.0225685468013881,0.0440075228376034,0.998775755508305],[0,0,0,0],[8.999999E+09,8.999999E+09,8.999999E+09,8.999999E+09,8.999999E+09,8.999999E+09]];
	LOCAL CONST Robtarget Tr_meulage_motif_1_P128 :=[[-47.4991015625,-92.257875,19.860359375],[-0.000994403231452177,0.0225685468013881,0.0440075228376034,0.998775755508305],[0,0,0,0],[8.999999E+09,8.999999E+09,8.999999E+09,8.999999E+09,8.999999E+09,8.999999E+09]];
	LOCAL CONST Robtarget Tr_meulage_motif_1_P129 :=[[-46.5098828125,-92.4038046875,19.8724140625],[-0.000994403231452177,0.0225685468013881,0.0440075228376034,0.998775755508305],[0,0,0,0],[8.999999E+09,8.999999E+09,8.999999E+09,8.999999E+09,8.999999E+09,8.999999E+09]];
	LOCAL CONST Robtarget Tr_meulage_motif_1_P130 :=[[-45.52066015625,-92.5497421875,19.884466796875],[-0.000994403231452177,0.0225685468013881,0.0440075228376034,0.998775755508305],[0,0,0,0],[8.999999E+09,8.999999E+09,8.999999E+09,8.999999E+09,8.999999E+09,8.999999E+09]];
	LOCAL CONST Robtarget Tr_meulage_motif_1_P131 :=[[-44.53144140625,-92.695671875,19.89651953125],[-0.000994403231452177,0.0225685468013881,0.0440075228376034,0.998775755508305],[0,0,0,0],[8.999999E+09,8.999999E+09,8.999999E+09,8.999999E+09,8.999999E+09,8.999999E+09]];
	LOCAL CONST Robtarget Tr_meulage_motif_1_P132 :=[[-43.54221875,-92.841609375,19.908572265625],[-0.000994403231452177,0.0225685468013881,0.0440075228376034,0.998775755508305],[0,0,0,0],[8.999999E+09,8.999999E+09,8.999999E+09,8.999999E+09,8.999999E+09,8.999999E+09]];
	LOCAL CONST Robtarget Tr_meulage_motif_1_P133 :=[[-42.55299609375,-92.9875390625,19.920626953125],[-0.000994403231452177,0.0225685468013881,0.0440075228376034,0.998775755508305],[0,0,0,0],[8.999999E+09,8.999999E+09,8.999999E+09,8.999999E+09,8.999999E+09,8.999999E+09]];
	LOCAL CONST Robtarget Tr_meulage_motif_1_P134 :=[[-41.56377734375,-93.1334765625,19.9326796875],[-0.000994403231452177,0.0225685468013881,0.0440075228376034,0.998775755508305],[0,0,0,0],[8.999999E+09,8.999999E+09,8.999999E+09,8.999999E+09,8.999999E+09,8.999999E+09]];
	LOCAL CONST Robtarget Tr_meulage_motif_1_P135 :=[[-40.56571875,-93.169375,19.9347109375],[-0.000994403231452177,0.0225685468013881,0.0440075228376034,0.998775755508305],[0,0,0,0],[8.999999E+09,8.999999E+09,8.999999E+09,8.999999E+09,8.999999E+09,8.999999E+09]];
	LOCAL CONST Robtarget Tr_meulage_motif_1_P136 :=[[-39.5788359375,-93.2056328125,19.936787109375],[-0.000994403231452177,0.0225685468013881,0.0440075228376034,0.998775755508305],[0,0,0,0],[8.999999E+09,8.999999E+09,8.999999E+09,8.999999E+09,8.999999E+09,8.999999E+09]];
	LOCAL CONST Robtarget Tr_meulage_motif_1_P137 :=[[-38.59727734375,-93.2430625,19.938978515625],[-0.000994403231452177,0.0225685468013881,0.0440075228376034,0.998775755508305],[0,0,0,0],[8.999999E+09,8.999999E+09,8.999999E+09,8.999999E+09,8.999999E+09,8.999999E+09]];
	LOCAL CONST Robtarget Tr_meulage_motif_1_P138 :=[[-37.6155078125,-93.2808046875,19.941197265625],[-0.000994403231452177,0.0225685468013881,0.0440075228376034,0.998775755508305],[0,0,0,0],[8.999999E+09,8.999999E+09,8.999999E+09,8.999999E+09,8.999999E+09,8.999999E+09]];
	LOCAL CONST Robtarget Tr_meulage_motif_1_P139 :=[[-36.4540859375,-93.2724375,19.938998046875],[-0.000994403231452177,0.0225685468013881,0.0440075228376034,0.998775755508305],[0,0,0,0],[8.999999E+09,8.999999E+09,8.999999E+09,8.999999E+09,8.999999E+09,8.999999E+09]];
	LOCAL CONST Robtarget Tr_meulage_motif_1_P140 :=[[-35.46819921875,-93.2288984375,19.933814453125],[-0.000994403231452177,0.0225685468013881,0.0440075228376034,0.998775755508305],[0,0,0,0],[8.999999E+09,8.999999E+09,8.999999E+09,8.999999E+09,8.999999E+09,8.999999E+09]];
	LOCAL CONST Robtarget Tr_meulage_motif_1_P141 :=[[-34.49420703125,-93.1529609375,19.92569921875],[-0.000994403231452177,0.0225685468013881,0.0440075228376034,0.998775755508305],[0,0,0,0],[8.999999E+09,8.999999E+09,8.999999E+09,8.999999E+09,8.999999E+09,8.999999E+09]];
	LOCAL CONST Robtarget Tr_meulage_motif_1_P142 :=[[-33.5158671875,-93.1055703125,19.92017578125],[-0.000994403231452177,0.0225685468013881,0.0440075228376034,0.998775755508305],[0,0,0,0],[8.999999E+09,8.999999E+09,8.999999E+09,8.999999E+09,8.999999E+09,8.999999E+09]];
	LOCAL CONST Robtarget Tr_meulage_motif_1_degg1 :=[[-33.9658103106873,-93.9850920946209,9.96909580867058],[-0.000994403231452177,0.0225685468013881,0.0440075228376034,0.998775755508305],[0,0,0,0],[8.999999E+09,8.999999E+09,8.999999E+09,8.999999E+09,8.999999E+09,8.999999E+09]];
	LOCAL CONST Robtarget Tr_meulage_motif_1_degg2 :=[[-42.5147296512452,-110.696005954918,-179.101423670339],[-0.000994403231452177,0.0225685468013881,0.0440075228376034,0.998775755508305],[0,0,0,0],[8.999999E+09,8.999999E+09,8.999999E+09,8.999999E+09,8.999999E+09,8.999999E+09]];
	LOCAL CONST Robtarget Tr_meulage_motif_2_App1 :=[[5.41975103712223,-169.550459000949,-174.452492700092],[-0.00047273798305717,0.0085506160566057,0.055200680935664,0.998438555098956],[0,0,0,0],[8.999999E+09,8.999999E+09,8.999999E+09,8.999999E+09,8.999999E+09,8.999999E+09]];
	LOCAL CONST Robtarget Tr_meulage_motif_2_App2 :=[[8.65399536435611,-148.605417481297,14.3618205798392],[-0.00047273798305717,0.0085506160566057,0.055200680935664,0.998438555098956],[0,0,0,0],[8.999999E+09,8.999999E+09,8.999999E+09,8.999999E+09,8.999999E+09,8.999999E+09]];
	LOCAL CONST Robtarget Tr_meulage_motif_2_P0 :=[[8.82421875,-147.503046875,24.299416015625],[-0.00047273798305717,0.0085506160566057,0.055200680935664,0.998438555098956],[0,0,0,0],[8.999999E+09,8.999999E+09,8.999999E+09,8.999999E+09,8.999999E+09,8.999999E+09]];
	LOCAL CONST Robtarget Tr_meulage_motif_2_P1 :=[[7.83119384765625,-147.385640625,24.288576171875],[-0.00047273798305717,0.0085506160566057,0.055200680935664,0.998438555098956],[0,0,0,0],[8.999999E+09,8.999999E+09,8.999999E+09,8.999999E+09,8.999999E+09,8.999999E+09]];
	LOCAL CONST Robtarget Tr_meulage_motif_2_P2 :=[[6.83816943359375,-147.268234375,24.27773828125],[-0.00047273798305717,0.0085506160566057,0.055200680935664,0.998438555098956],[0,0,0,0],[8.999999E+09,8.999999E+09,8.999999E+09,8.999999E+09,8.999999E+09,8.999999E+09]];
	LOCAL CONST Robtarget Tr_meulage_motif_2_P3 :=[[5.84514501953125,-147.150828125,24.266900390625],[-0.00047273798305717,0.0085506160566057,0.055200680935664,0.998438555098956],[0,0,0,0],[8.999999E+09,8.999999E+09,8.999999E+09,8.999999E+09,8.999999E+09,8.999999E+09]];
	LOCAL CONST Robtarget Tr_meulage_motif_2_P4 :=[[4.85212060546875,-147.033421875,24.256060546875],[-0.00047273798305717,0.0085506160566057,0.055200680935664,0.998438555098956],[0,0,0,0],[8.999999E+09,8.999999E+09,8.999999E+09,8.999999E+09,8.999999E+09,8.999999E+09]];
	LOCAL CONST Robtarget Tr_meulage_motif_2_P5 :=[[3.85909594726562,-146.916,24.24522265625],[-0.00047273798305717,0.0085506160566057,0.055200680935664,0.998438555098956],[0,0,0,0],[8.999999E+09,8.999999E+09,8.999999E+09,8.999999E+09,8.999999E+09,8.999999E+09]];
	LOCAL CONST Robtarget Tr_meulage_motif_2_P6 :=[[2.86607153320313,-146.79859375,24.234384765625],[-0.00047273798305717,0.0085506160566057,0.055200680935664,0.998438555098956],[0,0,0,0],[8.999999E+09,8.999999E+09,8.999999E+09,8.999999E+09,8.999999E+09,8.999999E+09]];
	LOCAL CONST Robtarget Tr_meulage_motif_2_P7 :=[[1.87304699707031,-146.6811875,24.223544921875],[-0.00047273798305717,0.0085506160566057,0.055200680935664,0.998438555098956],[0,0,0,0],[8.999999E+09,8.999999E+09,8.999999E+09,8.999999E+09,8.999999E+09,8.999999E+09]];
	LOCAL CONST Robtarget Tr_meulage_motif_2_P8 :=[[0.8800224609375,-146.56378125,24.21270703125],[-0.00047273798305717,0.0085506160566057,0.055200680935664,0.998438555098956],[0,0,0,0],[8.999999E+09,8.999999E+09,8.999999E+09,8.999999E+09,8.999999E+09,8.999999E+09]];
	LOCAL CONST Robtarget Tr_meulage_motif_2_P9 :=[[-0.113002029418945,-146.446375,24.201869140625],[-0.00047273798305717,0.0085506160566057,0.055200680935664,0.998438555098956],[0,0,0,0],[8.999999E+09,8.999999E+09,8.999999E+09,8.999999E+09,8.999999E+09,8.999999E+09]];
	LOCAL CONST Robtarget Tr_meulage_motif_2_P10 :=[[-1.10602648925781,-146.32896875,24.19103125],[-0.00047273798305717,0.0085506160566057,0.055200680935664,0.998438555098956],[0,0,0,0],[8.999999E+09,8.999999E+09,8.999999E+09,8.999999E+09,8.999999E+09,8.999999E+09]];
	LOCAL CONST Robtarget Tr_meulage_motif_2_P11 :=[[-2.09905102539062,-146.211546875,24.18019140625],[-0.00047273798305717,0.0085506160566057,0.055200680935664,0.998438555098956],[0,0,0,0],[8.999999E+09,8.999999E+09,8.999999E+09,8.999999E+09,8.999999E+09,8.999999E+09]];
	LOCAL CONST Robtarget Tr_meulage_motif_2_P12 :=[[-3.09207568359375,-146.094140625,24.169353515625],[-0.00047273798305717,0.0085506160566057,0.055200680935664,0.998438555098956],[0,0,0,0],[8.999999E+09,8.999999E+09,8.999999E+09,8.999999E+09,8.999999E+09,8.999999E+09]];
	LOCAL CONST Robtarget Tr_meulage_motif_2_P13 :=[[-4.08510009765625,-145.976734375,24.158515625],[-0.00047273798305717,0.0085506160566057,0.055200680935664,0.998438555098956],[0,0,0,0],[8.999999E+09,8.999999E+09,8.999999E+09,8.999999E+09,8.999999E+09,8.999999E+09]];
	LOCAL CONST Robtarget Tr_meulage_motif_2_P14 :=[[-5.07812451171875,-145.859328125,24.14767578125],[-0.00047273798305717,0.0085506160566057,0.055200680935664,0.998438555098956],[0,0,0,0],[8.999999E+09,8.999999E+09,8.999999E+09,8.999999E+09,8.999999E+09,8.999999E+09]];
	LOCAL CONST Robtarget Tr_meulage_motif_2_P15 :=[[-6.07114892578125,-145.741921875,24.136837890625],[-0.00047273798305717,0.0085506160566057,0.055200680935664,0.998438555098956],[0,0,0,0],[8.999999E+09,8.999999E+09,8.999999E+09,8.999999E+09,8.999999E+09,8.999999E+09]];
	LOCAL CONST Robtarget Tr_meulage_motif_2_P16 :=[[-7.064173828125,-145.624515625,24.126],[-0.00047273798305717,0.0085506160566057,0.055200680935664,0.998438555098956],[0,0,0,0],[8.999999E+09,8.999999E+09,8.999999E+09,8.999999E+09,8.999999E+09,8.999999E+09]];
	LOCAL CONST Robtarget Tr_meulage_motif_2_P17 :=[[-8.0571982421875,-145.50709375,24.115162109375],[-0.00047273798305717,0.0085506160566057,0.055200680935664,0.998438555098956],[0,0,0,0],[8.999999E+09,8.999999E+09,8.999999E+09,8.999999E+09,8.999999E+09,8.999999E+09]];
	LOCAL CONST Robtarget Tr_meulage_motif_2_P18 :=[[-9.05022265625,-145.3896875,24.104322265625],[-0.00047273798305717,0.0085506160566057,0.055200680935664,0.998438555098956],[0,0,0,0],[8.999999E+09,8.999999E+09,8.999999E+09,8.999999E+09,8.999999E+09,8.999999E+09]];
	LOCAL CONST Robtarget Tr_meulage_motif_2_P19 :=[[-10.022822265625,-145.16390625,24.08229296875],[-0.00047273798305717,0.0085506160566057,0.055200680935664,0.998438555098956],[0,0,0,0],[8.999999E+09,8.999999E+09,8.999999E+09,8.999999E+09,8.999999E+09,8.999999E+09]];
	LOCAL CONST Robtarget Tr_meulage_motif_2_P20 :=[[-10.9378203125,-144.844171875,24.050509765625],[-0.00047273798305717,0.0085506160566057,0.055200680935664,0.998438555098956],[0,0,0,0],[8.999999E+09,8.999999E+09,8.999999E+09,8.999999E+09,8.999999E+09,8.999999E+09]];
	LOCAL CONST Robtarget Tr_meulage_motif_2_P21 :=[[-11.752541015625,-144.475546875,24.013560546875],[-0.00047273798305717,0.0085506160566057,0.055200680935664,0.998438555098956],[0,0,0,0],[8.999999E+09,8.999999E+09,8.999999E+09,8.999999E+09,8.999999E+09,8.999999E+09]];
	LOCAL CONST Robtarget Tr_meulage_motif_2_P22 :=[[-12.4647138671875,-144.114921875,23.977306640625],[-0.00047273798305717,0.0085506160566057,0.055200680935664,0.998438555098956],[0,0,0,0],[8.999999E+09,8.999999E+09,8.999999E+09,8.999999E+09,8.999999E+09,8.999999E+09]];
	LOCAL CONST Robtarget Tr_meulage_motif_2_P23 :=[[-13.4854541015625,-143.377046875,23.902576171875],[-0.00047273798305717,0.0085506160566057,0.055200680935664,0.998438555098956],[0,0,0,0],[8.999999E+09,8.999999E+09,8.999999E+09,8.999999E+09,8.999999E+09,8.999999E+09]];
	LOCAL CONST Robtarget Tr_meulage_motif_2_P24 :=[[-14.4022470703125,-142.419546875,23.80508203125],[-0.00047273798305717,0.0085506160566057,0.055200680935664,0.998438555098956],[0,0,0,0],[8.999999E+09,8.999999E+09,8.999999E+09,8.999999E+09,8.999999E+09,8.999999E+09]];
	LOCAL CONST Robtarget Tr_meulage_motif_2_P25 :=[[-15.1232744140625,-141.30865625,23.691537109375],[-0.00047273798305717,0.0085506160566057,0.055200680935664,0.998438555098956],[0,0,0,0],[8.999999E+09,8.999999E+09,8.999999E+09,8.999999E+09,8.999999E+09,8.999999E+09]];
	LOCAL CONST Robtarget Tr_meulage_motif_2_P26 :=[[-15.4764248046875,-140.148796875,23.57248046875],[-0.00047273798305717,0.0085506160566057,0.055200680935664,0.998438555098956],[0,0,0,0],[8.999999E+09,8.999999E+09,8.999999E+09,8.999999E+09,8.999999E+09,8.999999E+09]];
	LOCAL CONST Robtarget Tr_meulage_motif_2_P27 :=[[-15.4212431640625,-139.45815625,23.501251953125],[-0.00047273798305717,0.0085506160566057,0.055200680935664,0.998438555098956],[0,0,0,0],[8.999999E+09,8.999999E+09,8.999999E+09,8.999999E+09,8.999999E+09,8.999999E+09]];
	LOCAL CONST Robtarget Tr_meulage_motif_2_P28 :=[[-15.34328125,-138.804984375,23.43385546875],[-0.00047273798305717,0.0085506160566057,0.055200680935664,0.998438555098956],[0,0,0,0],[8.999999E+09,8.999999E+09,8.999999E+09,8.999999E+09,8.999999E+09,8.999999E+09]];
	LOCAL CONST Robtarget Tr_meulage_motif_2_P29 :=[[-15.2108447265625,-138.15840625,23.367068359375],[-0.00047273798305717,0.0085506160566057,0.055200680935664,0.998438555098956],[0,0,0,0],[8.999999E+09,8.999999E+09,8.999999E+09,8.999999E+09,8.999999E+09,8.999999E+09]];
	LOCAL CONST Robtarget Tr_meulage_motif_2_P30 :=[[-14.586203125,-137.128609375,23.26017578125],[-0.00047273798305717,0.0085506160566057,0.055200680935664,0.998438555098956],[0,0,0,0],[8.999999E+09,8.999999E+09,8.999999E+09,8.999999E+09,8.999999E+09,8.999999E+09]];
	LOCAL CONST Robtarget Tr_meulage_motif_2_P31 :=[[-13.61687109375,-136.234875,23.166861328125],[-0.00047273798305717,0.0085506160566057,0.055200680935664,0.998438555098956],[0,0,0,0],[8.999999E+09,8.999999E+09,8.999999E+09,8.999999E+09,8.999999E+09,8.999999E+09]];
	LOCAL CONST Robtarget Tr_meulage_motif_2_P32 :=[[-12.50287890625,-135.53628125,23.093470703125],[-0.00047273798305717,0.0085506160566057,0.055200680935664,0.998438555098956],[0,0,0,0],[8.999999E+09,8.999999E+09,8.999999E+09,8.999999E+09,8.999999E+09,8.999999E+09]];
	LOCAL CONST Robtarget Tr_meulage_motif_2_P33 :=[[-11.77391796875,-135.22603125,23.06058203125],[-0.00047273798305717,0.0085506160566057,0.055200680935664,0.998438555098956],[0,0,0,0],[8.999999E+09,8.999999E+09,8.999999E+09,8.999999E+09,8.999999E+09,8.999999E+09]];
	LOCAL CONST Robtarget Tr_meulage_motif_2_P34 :=[[-10.5663603515625,-134.8804375,23.023443359375],[-0.00047273798305717,0.0085506160566057,0.055200680935664,0.998438555098956],[0,0,0,0],[8.999999E+09,8.999999E+09,8.999999E+09,8.999999E+09,8.999999E+09,8.999999E+09]];
	LOCAL CONST Robtarget Tr_meulage_motif_2_P35 :=[[-9.6960859375,-134.71878125,23.005685546875],[-0.00047273798305717,0.0085506160566057,0.055200680935664,0.998438555098956],[0,0,0,0],[8.999999E+09,8.999999E+09,8.999999E+09,8.999999E+09,8.999999E+09,8.999999E+09]];
	LOCAL CONST Robtarget Tr_meulage_motif_2_P36 :=[[-8.74648046875,-134.626234375,22.9949453125],[-0.00047273798305717,0.0085506160566057,0.055200680935664,0.998438555098956],[0,0,0,0],[8.999999E+09,8.999999E+09,8.999999E+09,8.999999E+09,8.999999E+09,8.999999E+09]];
	LOCAL CONST Robtarget Tr_meulage_motif_2_P37 :=[[-7.75896142578125,-134.63421875,22.994515625],[-0.00047273798305717,0.0085506160566057,0.055200680935664,0.998438555098956],[0,0,0,0],[8.999999E+09,8.999999E+09,8.999999E+09,8.999999E+09,8.999999E+09,8.999999E+09]];
	LOCAL CONST Robtarget Tr_meulage_motif_2_P38 :=[[-6.760283203125,-134.641515625,22.994001953125],[-0.00047273798305717,0.0085506160566057,0.055200680935664,0.998438555098956],[0,0,0,0],[8.999999E+09,8.999999E+09,8.999999E+09,8.999999E+09,8.999999E+09,8.999999E+09]];
	LOCAL CONST Robtarget Tr_meulage_motif_2_P39 :=[[-5.7672587890625,-134.758921875,23.00483984375],[-0.00047273798305717,0.0085506160566057,0.055200680935664,0.998438555098956],[0,0,0,0],[8.999999E+09,8.999999E+09,8.999999E+09,8.999999E+09,8.999999E+09,8.999999E+09]];
	LOCAL CONST Robtarget Tr_meulage_motif_2_P40 :=[[-4.774234375,-134.876328125,23.0156796875],[-0.00047273798305717,0.0085506160566057,0.055200680935664,0.998438555098956],[0,0,0,0],[8.999999E+09,8.999999E+09,8.999999E+09,8.999999E+09,8.999999E+09,8.999999E+09]];
	LOCAL CONST Robtarget Tr_meulage_motif_2_P41 :=[[-3.78120971679688,-134.993734375,23.026517578125],[-0.00047273798305717,0.0085506160566057,0.055200680935664,0.998438555098956],[0,0,0,0],[8.999999E+09,8.999999E+09,8.999999E+09,8.999999E+09,8.999999E+09,8.999999E+09]];
	LOCAL CONST Robtarget Tr_meulage_motif_2_P42 :=[[-2.78818505859375,-135.111140625,23.03735546875],[-0.00047273798305717,0.0085506160566057,0.055200680935664,0.998438555098956],[0,0,0,0],[8.999999E+09,8.999999E+09,8.999999E+09,8.999999E+09,8.999999E+09,8.999999E+09]];
	LOCAL CONST Robtarget Tr_meulage_motif_2_P43 :=[[-1.79516064453125,-135.2285625,23.0481953125],[-0.00047273798305717,0.0085506160566057,0.055200680935664,0.998438555098956],[0,0,0,0],[8.999999E+09,8.999999E+09,8.999999E+09,8.999999E+09,8.999999E+09,8.999999E+09]];
	LOCAL CONST Robtarget Tr_meulage_motif_2_P44 :=[[-0.802136108398438,-135.34596875,23.059033203125],[-0.00047273798305717,0.0085506160566057,0.055200680935664,0.998438555098956],[0,0,0,0],[8.999999E+09,8.999999E+09,8.999999E+09,8.999999E+09,8.999999E+09,8.999999E+09]];
	LOCAL CONST Robtarget Tr_meulage_motif_2_P45 :=[[0.190888397216797,-135.463375,23.06987109375],[-0.00047273798305717,0.0085506160566057,0.055200680935664,0.998438555098956],[0,0,0,0],[8.999999E+09,8.999999E+09,8.999999E+09,8.999999E+09,8.999999E+09,8.999999E+09]];
	LOCAL CONST Robtarget Tr_meulage_motif_2_P46 :=[[1.18391296386719,-135.58078125,23.080708984375],[-0.00047273798305717,0.0085506160566057,0.055200680935664,0.998438555098956],[0,0,0,0],[8.999999E+09,8.999999E+09,8.999999E+09,8.999999E+09,8.999999E+09,8.999999E+09]];
	LOCAL CONST Robtarget Tr_meulage_motif_2_P47 :=[[2.1769375,-135.6981875,23.091548828125],[-0.00047273798305717,0.0085506160566057,0.055200680935664,0.998438555098956],[0,0,0,0],[8.999999E+09,8.999999E+09,8.999999E+09,8.999999E+09,8.999999E+09,8.999999E+09]];
	LOCAL CONST Robtarget Tr_meulage_motif_2_P48 :=[[3.1699619140625,-135.81559375,23.10238671875],[-0.00047273798305717,0.0085506160566057,0.055200680935664,0.998438555098956],[0,0,0,0],[8.999999E+09,8.999999E+09,8.999999E+09,8.999999E+09,8.999999E+09,8.999999E+09]];
	LOCAL CONST Robtarget Tr_meulage_motif_2_P49 :=[[4.16864013671875,-135.822890625,23.101873046875],[-0.00047273798305717,0.0085506160566057,0.055200680935664,0.998438555098956],[0,0,0,0],[8.999999E+09,8.999999E+09,8.999999E+09,8.999999E+09,8.999999E+09,8.999999E+09]];
	LOCAL CONST Robtarget Tr_meulage_motif_2_P50 :=[[5.13343701171875,-135.72540625,23.09060546875],[-0.00047273798305717,0.0085506160566057,0.055200680935664,0.998438555098956],[0,0,0,0],[8.999999E+09,8.999999E+09,8.999999E+09,8.999999E+09,8.999999E+09,8.999999E+09]];
	LOCAL CONST Robtarget Tr_meulage_motif_2_P51 :=[[6.01225830078125,-135.557015625,23.072140625],[-0.00047273798305717,0.0085506160566057,0.055200680935664,0.998438555098956],[0,0,0,0],[8.999999E+09,8.999999E+09,8.999999E+09,8.999999E+09,8.999999E+09,8.999999E+09]];
	LOCAL CONST Robtarget Tr_meulage_motif_2_P52 :=[[6.75465576171875,-135.340109375,23.0488515625],[-0.00047273798305717,0.0085506160566057,0.055200680935664,0.998438555098956],[0,0,0,0],[8.999999E+09,8.999999E+09,8.999999E+09,8.999999E+09,8.999999E+09,8.999999E+09]];
	LOCAL CONST Robtarget Tr_meulage_motif_2_P53 :=[[7.86002197265625,-134.807125,22.992537109375],[-0.00047273798305717,0.0085506160566057,0.055200680935664,0.998438555098956],[0,0,0,0],[8.999999E+09,8.999999E+09,8.999999E+09,8.999999E+09,8.999999E+09,8.999999E+09]];
	LOCAL CONST Robtarget Tr_meulage_motif_2_P54 :=[[8.8620078125,-134.022109375,22.9103828125],[-0.00047273798305717,0.0085506160566057,0.055200680935664,0.998438555098956],[0,0,0,0],[8.999999E+09,8.999999E+09,8.999999E+09,8.999999E+09,8.999999E+09,8.999999E+09]];
	LOCAL CONST Robtarget Tr_meulage_motif_2_P55 :=[[9.5165732421875,-133.051671875,22.80956640625],[-0.00047273798305717,0.0085506160566057,0.055200680935664,0.998438555098956],[0,0,0,0],[8.999999E+09,8.999999E+09,8.999999E+09,8.999999E+09,8.999999E+09,8.999999E+09]];
	LOCAL CONST Robtarget Tr_meulage_motif_2_P56 :=[[9.781796875,-132.388609375,22.7409140625],[-0.00047273798305717,0.0085506160566057,0.055200680935664,0.998438555098956],[0,0,0,0],[8.999999E+09,8.999999E+09,8.999999E+09,8.999999E+09,8.999999E+09,8.999999E+09]];
	LOCAL CONST Robtarget Tr_meulage_motif_2_P57 :=[[9.9359794921875,-131.635515625,22.663125],[-0.00047273798305717,0.0085506160566057,0.055200680935664,0.998438555098956],[0,0,0,0],[8.999999E+09,8.999999E+09,8.999999E+09,8.999999E+09,8.999999E+09,8.999999E+09]];
	LOCAL CONST Robtarget Tr_meulage_motif_2_P58 :=[[9.9602783203125,-130.8671875,22.583931640625],[-0.00047273798305717,0.0085506160566057,0.055200680935664,0.998438555098956],[0,0,0,0],[8.999999E+09,8.999999E+09,8.999999E+09,8.999999E+09,8.999999E+09,8.999999E+09]];
	LOCAL CONST Robtarget Tr_meulage_motif_2_P59 :=[[9.674275390625,-129.72321875,22.46642578125],[-0.00047273798305717,0.0085506160566057,0.055200680935664,0.998438555098956],[0,0,0,0],[8.999999E+09,8.999999E+09,8.999999E+09,8.999999E+09,8.999999E+09,8.999999E+09]];
	LOCAL CONST Robtarget Tr_meulage_motif_2_P60 :=[[9.33190625,-129.0960390625,22.402240234375],[-0.00047273798305717,0.0085506160566057,0.055200680935664,0.998438555098956],[0,0,0,0],[8.999999E+09,8.999999E+09,8.999999E+09,8.999999E+09,8.999999E+09,8.999999E+09]];
	LOCAL CONST Robtarget Tr_meulage_motif_2_P61 :=[[8.5555625,-128.1156015625,22.30220703125],[-0.00047273798305717,0.0085506160566057,0.055200680935664,0.998438555098956],[0,0,0,0],[8.999999E+09,8.999999E+09,8.999999E+09,8.999999E+09,8.999999E+09,8.999999E+09]];
	LOCAL CONST Robtarget Tr_meulage_motif_2_P62 :=[[8.02280859375,-127.6375859375,22.253630859375],[-0.00047273798305717,0.0085506160566057,0.055200680935664,0.998438555098956],[0,0,0,0],[8.999999E+09,8.999999E+09,8.999999E+09,8.999999E+09,8.999999E+09,8.999999E+09]];
	LOCAL CONST Robtarget Tr_meulage_motif_2_P63 :=[[6.976849609375,-126.968890625,22.18605859375],[-0.00047273798305717,0.0085506160566057,0.055200680935664,0.998438555098956],[0,0,0,0],[8.999999E+09,8.999999E+09,8.999999E+09,8.999999E+09,8.999999E+09,8.999999E+09]];
	LOCAL CONST Robtarget Tr_meulage_motif_2_P64 :=[[6.1918544921875,-126.5800703125,22.1469921875],[-0.00047273798305717,0.0085506160566057,0.055200680935664,0.998438555098956],[0,0,0,0],[8.999999E+09,8.999999E+09,8.999999E+09,8.999999E+09,8.999999E+09,8.999999E+09]];
	LOCAL CONST Robtarget Tr_meulage_motif_2_P65 :=[[5.290462890625,-126.268671875,22.116048828125],[-0.00047273798305717,0.0085506160566057,0.055200680935664,0.998438555098956],[0,0,0,0],[8.999999E+09,8.999999E+09,8.999999E+09,8.999999E+09,8.999999E+09,8.999999E+09]];
	LOCAL CONST Robtarget Tr_meulage_motif_2_P66 :=[[4.32855078125,-126.0461640625,22.094341796875],[-0.00047273798305717,0.0085506160566057,0.055200680935664,0.998438555098956],[0,0,0,0],[8.999999E+09,8.999999E+09,8.999999E+09,8.999999E+09,8.999999E+09,8.999999E+09]];
	LOCAL CONST Robtarget Tr_meulage_motif_2_P67 :=[[3.35595092773438,-125.8203828125,22.0723125],[-0.00047273798305717,0.0085506160566057,0.055200680935664,0.998438555098956],[0,0,0,0],[8.999999E+09,8.999999E+09,8.999999E+09,8.999999E+09,8.999999E+09,8.999999E+09]];
	LOCAL CONST Robtarget Tr_meulage_motif_2_P68 :=[[2.36292651367188,-125.7029765625,22.061474609375],[-0.00047273798305717,0.0085506160566057,0.055200680935664,0.998438555098956],[0,0,0,0],[8.999999E+09,8.999999E+09,8.999999E+09,8.999999E+09,8.999999E+09,8.999999E+09]];
	LOCAL CONST Robtarget Tr_meulage_motif_2_P69 :=[[1.36990197753906,-125.5855625,22.05063671875],[-0.00047273798305717,0.0085506160566057,0.055200680935664,0.998438555098956],[0,0,0,0],[8.999999E+09,8.999999E+09,8.999999E+09,8.999999E+09,8.999999E+09,8.999999E+09]];
	LOCAL CONST Robtarget Tr_meulage_motif_2_P70 :=[[0.37687744140625,-125.46815625,22.039796875],[-0.00047273798305717,0.0085506160566057,0.055200680935664,0.998438555098956],[0,0,0,0],[8.999999E+09,8.999999E+09,8.999999E+09,8.999999E+09,8.999999E+09,8.999999E+09]];
	LOCAL CONST Robtarget Tr_meulage_motif_2_P71 :=[[-0.616147033691406,-125.35075,22.028958984375],[-0.00047273798305717,0.0085506160566057,0.055200680935664,0.998438555098956],[0,0,0,0],[8.999999E+09,8.999999E+09,8.999999E+09,8.999999E+09,8.999999E+09,8.999999E+09]];
	LOCAL CONST Robtarget Tr_meulage_motif_2_P72 :=[[-1.60917150878906,-125.2333359375,22.01812109375],[-0.00047273798305717,0.0085506160566057,0.055200680935664,0.998438555098956],[0,0,0,0],[8.999999E+09,8.999999E+09,8.999999E+09,8.999999E+09,8.999999E+09,8.999999E+09]];
	LOCAL CONST Robtarget Tr_meulage_motif_2_P73 :=[[-2.60219604492187,-125.1159296875,22.00728125],[-0.00047273798305717,0.0085506160566057,0.055200680935664,0.998438555098956],[0,0,0,0],[8.999999E+09,8.999999E+09,8.999999E+09,8.999999E+09,8.999999E+09,8.999999E+09]];
	LOCAL CONST Robtarget Tr_meulage_motif_2_P74 :=[[-3.595220703125,-124.9985234375,21.996443359375],[-0.00047273798305717,0.0085506160566057,0.055200680935664,0.998438555098956],[0,0,0,0],[8.999999E+09,8.999999E+09,8.999999E+09,8.999999E+09,8.999999E+09,8.999999E+09]];
	LOCAL CONST Robtarget Tr_meulage_motif_2_P75 :=[[-4.5882451171875,-124.881109375,21.98560546875],[-0.00047273798305717,0.0085506160566057,0.055200680935664,0.998438555098956],[0,0,0,0],[8.999999E+09,8.999999E+09,8.999999E+09,8.999999E+09,8.999999E+09,8.999999E+09]];
	LOCAL CONST Robtarget Tr_meulage_motif_2_P76 :=[[-5.58126953125,-124.763703125,21.974765625],[-0.00047273798305717,0.0085506160566057,0.055200680935664,0.998438555098956],[0,0,0,0],[8.999999E+09,8.999999E+09,8.999999E+09,8.999999E+09,8.999999E+09,8.999999E+09]];
	LOCAL CONST Robtarget Tr_meulage_motif_2_P77 :=[[-6.5742939453125,-124.646296875,21.963927734375],[-0.00047273798305717,0.0085506160566057,0.055200680935664,0.998438555098956],[0,0,0,0],[8.999999E+09,8.999999E+09,8.999999E+09,8.999999E+09,8.999999E+09,8.999999E+09]];
	LOCAL CONST Robtarget Tr_meulage_motif_2_P78 :=[[-7.54689404296875,-124.420515625,21.9418984375],[-0.00047273798305717,0.0085506160566057,0.055200680935664,0.998438555098956],[0,0,0,0],[8.999999E+09,8.999999E+09,8.999999E+09,8.999999E+09,8.999999E+09,8.999999E+09]];
	LOCAL CONST Robtarget Tr_meulage_motif_2_P79 :=[[-8.461892578125,-124.10078125,21.910115234375],[-0.00047273798305717,0.0085506160566057,0.055200680935664,0.998438555098956],[0,0,0,0],[8.999999E+09,8.999999E+09,8.999999E+09,8.999999E+09,8.999999E+09,8.999999E+09]];
	LOCAL CONST Robtarget Tr_meulage_motif_2_P80 :=[[-9.2766123046875,-123.732140625,21.873166015625],[-0.00047273798305717,0.0085506160566057,0.055200680935664,0.998438555098956],[0,0,0,0],[8.999999E+09,8.999999E+09,8.999999E+09,8.999999E+09,8.999999E+09,8.999999E+09]];
	LOCAL CONST Robtarget Tr_meulage_motif_2_P81 :=[[-9.98878515625,-123.37153125,21.836912109375],[-0.00047273798305717,0.0085506160566057,0.055200680935664,0.998438555098956],[0,0,0,0],[8.999999E+09,8.999999E+09,8.999999E+09,8.999999E+09,8.999999E+09,8.999999E+09]];
	LOCAL CONST Robtarget Tr_meulage_motif_2_P82 :=[[-11.009525390625,-122.63365625,21.762181640625],[-0.00047273798305717,0.0085506160566057,0.055200680935664,0.998438555098956],[0,0,0,0],[8.999999E+09,8.999999E+09,8.999999E+09,8.999999E+09,8.999999E+09,8.999999E+09]];
	LOCAL CONST Robtarget Tr_meulage_motif_2_P83 :=[[-11.854169921875,-121.63828125,21.6606953125],[-0.00047273798305717,0.0085506160566057,0.055200680935664,0.998438555098956],[0,0,0,0],[8.999999E+09,8.999999E+09,8.999999E+09,8.999999E+09,8.999999E+09,8.999999E+09]];
	LOCAL CONST Robtarget Tr_meulage_motif_2_P84 :=[[-12.3310048828125,-120.4940390625,21.543404296875],[-0.00047273798305717,0.0085506160566057,0.055200680935664,0.998438555098956],[0,0,0,0],[8.999999E+09,8.999999E+09,8.999999E+09,8.999999E+09,8.999999E+09,8.999999E+09]];
	LOCAL CONST Robtarget Tr_meulage_motif_2_P85 :=[[-12.383078125,-119.5018125,21.44123828125],[-0.00047273798305717,0.0085506160566057,0.055200680935664,0.998438555098956],[0,0,0,0],[8.999999E+09,8.999999E+09,8.999999E+09,8.999999E+09,8.999999E+09,8.999999E+09]];
	LOCAL CONST Robtarget Tr_meulage_motif_2_P86 :=[[-12.228396484375,-119.31509375,21.421802734375],[-0.00047273798305717,0.0085506160566057,0.055200680935664,0.998438555098956],[0,0,0,0],[8.999999E+09,8.999999E+09,8.999999E+09,8.999999E+09,8.999999E+09,8.999999E+09]];
	LOCAL CONST Robtarget Tr_meulage_motif_2_P87 :=[[-12.02023828125,-118.612046875,21.349103515625],[-0.00047273798305717,0.0085506160566057,0.055200680935664,0.998438555098956],[0,0,0,0],[8.999999E+09,8.999999E+09,8.999999E+09,8.999999E+09,8.999999E+09,8.999999E+09]];
	LOCAL CONST Robtarget Tr_meulage_motif_2_P88 :=[[-11.230546875,-117.7668984375,21.2610234375],[-0.00047273798305717,0.0085506160566057,0.055200680935664,0.998438555098956],[0,0,0,0],[8.999999E+09,8.999999E+09,8.999999E+09,8.999999E+09,8.999999E+09,8.999999E+09]];
	LOCAL CONST Robtarget Tr_meulage_motif_2_P89 :=[[-10.622126953125,-117.3742265625,21.219794921875],[-0.00047273798305717,0.0085506160566057,0.055200680935664,0.998438555098956],[0,0,0,0],[8.999999E+09,8.999999E+09,8.999999E+09,8.999999E+09,8.999999E+09,8.999999E+09]];
	LOCAL CONST Robtarget Tr_meulage_motif_2_P90 :=[[-9.43716015625,-116.9829765625,21.17798046875],[-0.00047273798305717,0.0085506160566057,0.055200680935664,0.998438555098956],[0,0,0,0],[8.999999E+09,8.999999E+09,8.999999E+09,8.999999E+09,8.999999E+09,8.999999E+09]];
	LOCAL CONST Robtarget Tr_meulage_motif_2_P91 :=[[-8.56688671875,-116.8213203125,21.16022265625],[-0.00047273798305717,0.0085506160566057,0.055200680935664,0.998438555098956],[0,0,0,0],[8.999999E+09,8.999999E+09,8.999999E+09,8.999999E+09,8.999999E+09,8.999999E+09]];
	LOCAL CONST Robtarget Tr_meulage_motif_2_P92 :=[[-7.6172802734375,-116.72878125,21.149484375],[-0.00047273798305717,0.0085506160566057,0.055200680935664,0.998438555098956],[0,0,0,0],[8.999999E+09,8.999999E+09,8.999999E+09,8.999999E+09,8.999999E+09,8.999999E+09]];
	LOCAL CONST Robtarget Tr_meulage_motif_2_P93 :=[[-6.62976123046875,-116.7367578125,21.1490546875],[-0.00047273798305717,0.0085506160566057,0.055200680935664,0.998438555098956],[0,0,0,0],[8.999999E+09,8.999999E+09,8.999999E+09,8.999999E+09,8.999999E+09,8.999999E+09]];
	LOCAL CONST Robtarget Tr_meulage_motif_2_P94 :=[[-5.63108349609375,-116.744046875,21.1485390625],[-0.00047273798305717,0.0085506160566057,0.055200680935664,0.998438555098956],[0,0,0,0],[8.999999E+09,8.999999E+09,8.999999E+09,8.999999E+09,8.999999E+09,8.999999E+09]];
	LOCAL CONST Robtarget Tr_meulage_motif_2_P95 :=[[-4.63805859375,-116.8614609375,21.15937890625],[-0.00047273798305717,0.0085506160566057,0.055200680935664,0.998438555098956],[0,0,0,0],[8.999999E+09,8.999999E+09,8.999999E+09,8.999999E+09,8.999999E+09,8.999999E+09]];
	LOCAL CONST Robtarget Tr_meulage_motif_2_P96 :=[[-3.6450341796875,-116.9788671875,21.170216796875],[-0.00047273798305717,0.0085506160566057,0.055200680935664,0.998438555098956],[0,0,0,0],[8.999999E+09,8.999999E+09,8.999999E+09,8.999999E+09,8.999999E+09,8.999999E+09]];
	LOCAL CONST Robtarget Tr_meulage_motif_2_P97 :=[[-2.652009765625,-117.0962734375,21.1810546875],[-0.00047273798305717,0.0085506160566057,0.055200680935664,0.998438555098956],[0,0,0,0],[8.999999E+09,8.999999E+09,8.999999E+09,8.999999E+09,8.999999E+09,8.999999E+09]];
	LOCAL CONST Robtarget Tr_meulage_motif_2_P98 :=[[-1.65898522949219,-117.2136875,21.191892578125],[-0.00047273798305717,0.0085506160566057,0.055200680935664,0.998438555098956],[0,0,0,0],[8.999999E+09,8.999999E+09,8.999999E+09,8.999999E+09,8.999999E+09,8.999999E+09]];
	LOCAL CONST Robtarget Tr_meulage_motif_2_P99 :=[[-0.665960693359375,-117.33109375,21.202732421875],[-0.00047273798305717,0.0085506160566057,0.055200680935664,0.998438555098956],[0,0,0,0],[8.999999E+09,8.999999E+09,8.999999E+09,8.999999E+09,8.999999E+09,8.999999E+09]];
	LOCAL CONST Robtarget Tr_meulage_motif_2_P100 :=[[0.327063812255859,-117.4485,21.2135703125],[-0.00047273798305717,0.0085506160566057,0.055200680935664,0.998438555098956],[0,0,0,0],[8.999999E+09,8.999999E+09,8.999999E+09,8.999999E+09,8.999999E+09,8.999999E+09]];
	LOCAL CONST Robtarget Tr_meulage_motif_2_P101 :=[[1.32008825683594,-117.5659140625,21.224408203125],[-0.00047273798305717,0.0085506160566057,0.055200680935664,0.998438555098956],[0,0,0,0],[8.999999E+09,8.999999E+09,8.999999E+09,8.999999E+09,8.999999E+09,8.999999E+09]];
	LOCAL CONST Robtarget Tr_meulage_motif_2_P102 :=[[2.31311279296875,-117.6833203125,21.235248046875],[-0.00047273798305717,0.0085506160566057,0.055200680935664,0.998438555098956],[0,0,0,0],[8.999999E+09,8.999999E+09,8.999999E+09,8.999999E+09,8.999999E+09,8.999999E+09]];
	LOCAL CONST Robtarget Tr_meulage_motif_2_P103 :=[[3.30613745117188,-117.8007265625,21.2460859375],[-0.00047273798305717,0.0085506160566057,0.055200680935664,0.998438555098956],[0,0,0,0],[8.999999E+09,8.999999E+09,8.999999E+09,8.999999E+09,8.999999E+09,8.999999E+09]];
	LOCAL CONST Robtarget Tr_meulage_motif_2_P104 :=[[4.29916162109375,-117.918140625,21.256923828125],[-0.00047273798305717,0.0085506160566057,0.055200680935664,0.998438555098956],[0,0,0,0],[8.999999E+09,8.999999E+09,8.999999E+09,8.999999E+09,8.999999E+09,8.999999E+09]];
	LOCAL CONST Robtarget Tr_meulage_motif_2_P105 :=[[5.2921865234375,-118.035546875,21.267763671875],[-0.00047273798305717,0.0085506160566057,0.055200680935664,0.998438555098956],[0,0,0,0],[8.999999E+09,8.999999E+09,8.999999E+09,8.999999E+09,8.999999E+09,8.999999E+09]];
	LOCAL CONST Robtarget Tr_meulage_motif_2_P106 :=[[6.2852109375,-118.152953125,21.2786015625],[-0.00047273798305717,0.0085506160566057,0.055200680935664,0.998438555098956],[0,0,0,0],[8.999999E+09,8.999999E+09,8.999999E+09,8.999999E+09,8.999999E+09,8.999999E+09]];
	LOCAL CONST Robtarget Tr_meulage_motif_2_P107 :=[[7.2782353515625,-118.2703671875,21.289439453125],[-0.00047273798305717,0.0085506160566057,0.055200680935664,0.998438555098956],[0,0,0,0],[8.999999E+09,8.999999E+09,8.999999E+09,8.999999E+09,8.999999E+09,8.999999E+09]];
	LOCAL CONST Robtarget Tr_meulage_motif_2_P108 :=[[8.271259765625,-118.3877734375,21.30027734375],[-0.00047273798305717,0.0085506160566057,0.055200680935664,0.998438555098956],[0,0,0,0],[8.999999E+09,8.999999E+09,8.999999E+09,8.999999E+09,8.999999E+09,8.999999E+09]];
	LOCAL CONST Robtarget Tr_meulage_motif_2_P109 :=[[9.2642841796875,-118.5051796875,21.3111171875],[-0.00047273798305717,0.0085506160566057,0.055200680935664,0.998438555098956],[0,0,0,0],[8.999999E+09,8.999999E+09,8.999999E+09,8.999999E+09,8.999999E+09,8.999999E+09]];
	LOCAL CONST Robtarget Tr_meulage_motif_2_P110 :=[[10.25730859375,-118.62259375,21.321955078125],[-0.00047273798305717,0.0085506160566057,0.055200680935664,0.998438555098956],[0,0,0,0],[8.999999E+09,8.999999E+09,8.999999E+09,8.999999E+09,8.999999E+09,8.999999E+09]];
	LOCAL CONST Robtarget Tr_meulage_motif_2_P111 :=[[11.2503330078125,-118.74,21.33279296875],[-0.00047273798305717,0.0085506160566057,0.055200680935664,0.998438555098956],[0,0,0,0],[8.999999E+09,8.999999E+09,8.999999E+09,8.999999E+09,8.999999E+09,8.999999E+09]];
	LOCAL CONST Robtarget Tr_meulage_motif_2_P112 :=[[12.2433583984375,-118.85740625,21.3436328125],[-0.00047273798305717,0.0085506160566057,0.055200680935664,0.998438555098956],[0,0,0,0],[8.999999E+09,8.999999E+09,8.999999E+09,8.999999E+09,8.999999E+09,8.999999E+09]];
	LOCAL CONST Robtarget Tr_meulage_motif_2_P113 :=[[13.2363828125,-118.9748203125,21.354470703125],[-0.00047273798305717,0.0085506160566057,0.055200680935664,0.998438555098956],[0,0,0,0],[8.999999E+09,8.999999E+09,8.999999E+09,8.999999E+09,8.999999E+09,8.999999E+09]];
	LOCAL CONST Robtarget Tr_meulage_motif_2_P114 :=[[14.2294072265625,-119.0922265625,21.36530859375],[-0.00047273798305717,0.0085506160566057,0.055200680935664,0.998438555098956],[0,0,0,0],[8.999999E+09,8.999999E+09,8.999999E+09,8.999999E+09,8.999999E+09,8.999999E+09]];
	LOCAL CONST Robtarget Tr_meulage_motif_2_P115 :=[[15.222431640625,-119.2096328125,21.376146484375],[-0.00047273798305717,0.0085506160566057,0.055200680935664,0.998438555098956],[0,0,0,0],[8.999999E+09,8.999999E+09,8.999999E+09,8.999999E+09,8.999999E+09,8.999999E+09]];
	LOCAL CONST Robtarget Tr_meulage_motif_2_degg1 :=[[15.0522082549811,-120.312003418797,11.4385510485892],[-0.00047273798305717,0.0085506160566057,0.055200680935664,0.998438555098956],[0,0,0,0],[8.999999E+09,8.999999E+09,8.999999E+09,8.999999E+09,8.999999E+09,8.999999E+09]];
	LOCAL CONST Robtarget Tr_meulage_motif_2_degg2 :=[[11.8179639277472,-141.257044938449,-177.375762231342],[-0.00047273798305717,0.0085506160566057,0.055200680935664,0.998438555098956],[0,0,0,0],[8.999999E+09,8.999999E+09,8.999999E+09,8.999999E+09,8.999999E+09,8.999999E+09]];
	LOCAL CONST Robtarget Tr_meulage_bavure_App1 :=[[329.544731806537,56.7586330740036,78.3868810915932],[0.557702104481969,-0.547510182831542,-0.437048849622104,0.445184529601098],[0,0,0,0],[8.999999E+09,8.999999E+09,8.999999E+09,8.999999E+09,8.999999E+09,8.999999E+09]];
	LOCAL CONST Robtarget Tr_meulage_bavure_App2 :=[[144.300003777827,98.8551070443252,81.8908241327047],[0.557702104481969,-0.547510182831542,-0.437048849622104,0.445184529601098],[0,0,0,0],[8.999999E+09,8.999999E+09,8.999999E+09,8.999999E+09,8.999999E+09,8.999999E+09]];
	LOCAL CONST Robtarget Tr_meulage_bavure_P0 :=[[134.55028125,101.0707109375,82.0752421875],[0.557702104481969,-0.547510182831542,-0.437048849622104,0.445184529601098],[0,0,0,0],[8.999999E+09,8.999999E+09,8.999999E+09,8.999999E+09,8.999999E+09,8.999999E+09]];
	LOCAL CONST Robtarget Tr_meulage_bavure_P1 :=[[134.524625,100.3267578125,82.1859140625],[0.558215141104453,-0.548024689618692,-0.436414858764422,0.44452993921636],[0,0,0,0],[8.999999E+09,8.999999E+09,8.999999E+09,8.999999E+09,8.999999E+09,8.999999E+09]];
	LOCAL CONST Robtarget Tr_meulage_bavure_P2 :=[[134.694515625,97.4322109375,82.608484375],[0.559653396987563,-0.549448670693033,-0.434633232700365,0.442705530286634],[0,0,0,0],[8.999999E+09,8.999999E+09,8.999999E+09,8.999999E+09,8.999999E+09,8.999999E+09]];
	LOCAL CONST Robtarget Tr_meulage_bavure_P3 :=[[134.586953125,96.8921484375,82.69146875],[0.561717836919846,-0.551492805161999,-0.432054728286668,0.440065301183555],[0,0,0,0],[8.999999E+09,8.999999E+09,8.999999E+09,8.999999E+09,8.999999E+09,8.999999E+09]];
	LOCAL CONST Robtarget Tr_meulage_bavure_P4 :=[[134.468671875,96.45815625,82.7590859375],[0.56406159855728,-0.553822151274322,-0.429094537670899,0.43702793449834],[0,0,0,0],[8.999999E+09,8.999999E+09,8.999999E+09,8.999999E+09,8.999999E+09,8.999999E+09]];
	LOCAL CONST Robtarget Tr_meulage_bavure_P5 :=[[133.704234375,93.9382109375,83.1540546875],[0.566335533710986,-0.556089033831523,-0.426188747769959,0.434041704197753],[0,0,0,0],[8.999999E+09,8.999999E+09,8.999999E+09,8.999999E+09,8.999999E+09,8.999999E+09]];
	LOCAL CONST Robtarget Tr_meulage_bavure_P6 :=[[131.725109375,87.7298125,84.1299765625],[0.568254050492895,-0.558020170995036,-0.423707149902689,0.431477779245269],[0,0,0,0],[8.999999E+09,8.999999E+09,8.999999E+09,8.999999E+09,8.999999E+09,8.999999E+09]];
	LOCAL CONST Robtarget Tr_meulage_bavure_P7 :=[[131.510359375,87.1313515625,84.2247578125],[0.56969117307832,-0.559483621544917,-0.421828143819746,0.429524227048045],[0,0,0,0],[8.999999E+09,8.999999E+09,8.999999E+09,8.999999E+09,8.999999E+09,8.999999E+09]];
	LOCAL CONST Robtarget Tr_meulage_bavure_P8 :=[[131.3601875,86.625296875,84.3039765625],[0.570585548500341,-0.560430260951484,-0.420642054322016,0.428264306927593],[0,0,0,0],[8.999999E+09,8.999999E+09,8.999999E+09,8.999999E+09,8.999999E+09,8.999999E+09]];
	LOCAL CONST Robtarget Tr_meulage_bavure_P9 :=[[128.3930078125,76.715703125,85.8560078125],[0.570983810130519,-0.560891075904192,-0.420101275175689,0.427660622615215],[0,0,0,0],[8.999999E+09,8.999999E+09,8.999999E+09,8.999999E+09,8.999999E+09,8.999999E+09]];
	LOCAL CONST Robtarget Tr_meulage_bavure_P10 :=[[128.01440625,75.5305234375,86.0423359375],[0.571003066209651,-0.560999209584174,-0.420051503462695,0.427541950764878],[0,0,0,0],[8.999999E+09,8.999999E+09,8.999999E+09,8.999999E+09,8.999999E+09,8.999999E+09]];
	LOCAL CONST Robtarget Tr_meulage_bavure_P11 :=[[126.226359375,69.7393828125,86.9509375],[0.570740801955338,-0.560842065218131,-0.420367882558587,0.427787281459429],[0,0,0,0],[8.999999E+09,8.999999E+09,8.999999E+09,8.999999E+09,8.999999E+09,8.999999E+09]];
	LOCAL CONST Robtarget Tr_meulage_bavure_P12 :=[[125.3141640625,66.648265625,87.434671875],[0.57033794948801,-0.560557484353795,-0.420865213397034,0.428208363137651],[0,0,0,0],[8.999999E+09,8.999999E+09,8.999999E+09,8.999999E+09,8.999999E+09,8.999999E+09]];
	LOCAL CONST Robtarget Tr_meulage_bavure_P13 :=[[124.012546875,62.1365546875,88.139828125],[0.569899216368102,-0.560255944543128,-0.421403844970475,0.428657158147639],[0,0,0,0],[8.999999E+09,8.999999E+09,8.999999E+09,8.999999E+09,8.999999E+09,8.999999E+09]];
	LOCAL CONST Robtarget Tr_meulage_bavure_P14 :=[[122.837,57.78696484375,88.8172890625],[0.569547296799522,-0.560045255139164,-0.421826964339989,0.42898391701808],[0,0,0,0],[8.999999E+09,8.999999E+09,8.999999E+09,8.999999E+09,8.999999E+09,8.999999E+09]];
	LOCAL CONST Robtarget Tr_meulage_bavure_P15 :=[[121.8086640625,54.39926171875,89.34828125],[0.569353669037561,-0.560010274071851,-0.422037807812043,0.429079224927802],[0,0,0,0],[8.999999E+09,8.999999E+09,8.999999E+09,8.999999E+09,8.999999E+09,8.999999E+09]];
	LOCAL CONST Robtarget Tr_meulage_bavure_P16 :=[[119.8079453125,47.48033203125,90.4298125],[0.569403538493391,-0.560221592174139,-0.421928894411092,0.428844244538867],[0,0,0,0],[8.999999E+09,8.999999E+09,8.999999E+09,8.999999E+09,8.999999E+09,8.999999E+09]];
	LOCAL CONST Robtarget Tr_meulage_bavure_P17 :=[[118.310796875,41.38067578125,91.375359375],[0.569692926971746,-0.560691002259953,-0.421500303269638,0.428267513695233],[0,0,0,0],[8.999999E+09,8.999999E+09,8.999999E+09,8.999999E+09,8.999999E+09,8.999999E+09]];
	LOCAL CONST Robtarget Tr_meulage_bavure_P18 :=[[117.5947890625,38.56939453125,91.8119296875],[0.570233125924566,-0.561413731723629,-0.420739443859568,0.427348949116748],[0,0,0,0],[8.999999E+09,8.999999E+09,8.999999E+09,8.999999E+09,8.999999E+09,8.999999E+09]];
	LOCAL CONST Robtarget Tr_meulage_bavure_P19 :=[[117.0188359375,36.155328125,92.18565625],[0.570971212702887,-0.562348725357408,-0.419709643042559,0.426145046774665],[0,0,0,0],[8.999999E+09,8.999999E+09,8.999999E+09,8.999999E+09,8.999999E+09,8.999999E+09]];
	LOCAL CONST Robtarget Tr_meulage_bavure_P20 :=[[116.4451640625,34.09753125,92.5066875],[0.571838923568948,-0.563421479228843,-0.418499814741366,0.424752148077595],[0,0,0,0],[8.999999E+09,8.999999E+09,8.999999E+09,8.999999E+09,8.999999E+09,8.999999E+09]];
	LOCAL CONST Robtarget Tr_meulage_bavure_P21 :=[[115.1916328125,29.72143359375,93.1903828125],[0.572754406527106,-0.564551994789841,-0.417216108748344,0.423277868052989],[0,0,0,0],[8.999999E+09,8.999999E+09,8.999999E+09,8.999999E+09,8.999999E+09,8.999999E+09]];
	LOCAL CONST Robtarget Tr_meulage_bavure_P22 :=[[114.5182578125,27.486966796875,93.54046875],[0.573638385682801,-0.565661920368146,-0.415963626420593,0.421829178473562],[0,0,0,0],[8.999999E+09,8.999999E+09,8.999999E+09,8.999999E+09,8.999999E+09,8.999999E+09]];
	LOCAL CONST Robtarget Tr_meulage_bavure_P23 :=[[113.1544140625,23.533318359375,94.1650234375],[0.574428723905919,-0.566686714888883,-0.414827532714971,0.420494858971991],[0,0,0,0],[8.999999E+09,8.999999E+09,8.999999E+09,8.999999E+09,8.999999E+09,8.999999E+09]];
	LOCAL CONST Robtarget Tr_meulage_bavure_P24 :=[[112.753875,22.310947265625,94.3575],[0.575086137406628,-0.567584581704442,-0.413863616932666,0.419333499441112],[0,0,0,0],[8.999999E+09,8.999999E+09,8.999999E+09,8.999999E+09,8.999999E+09,8.999999E+09]];
	LOCAL CONST Robtarget Tr_meulage_bavure_P25 :=[[112.5212109375,21.7902265625,94.441328125],[0.575593769631112,-0.568345034959706,-0.413095061902639,0.418363721455568],[0,0,0,0],[8.999999E+09,8.999999E+09,8.999999E+09,8.999999E+09,8.999999E+09,8.999999E+09]];
	LOCAL CONST Robtarget Tr_meulage_bavure_P26 :=[[111.425296875,16.677486328125,95.229171875],[0.575966845401685,-0.568968959059754,-0.412507597674846,0.417581128027859],[0,0,0,0],[8.999999E+09,8.999999E+09,8.999999E+09,8.999999E+09,8.999999E+09,8.999999E+09]];
	LOCAL CONST Robtarget Tr_meulage_bavure_P27 :=[[111.212796875,15.838138671875,95.3594765625],[0.576220525941713,-0.56948133362122,-0.412078951554155,0.416955457844698],[0,0,0,0],[8.999999E+09,8.999999E+09,8.999999E+09,8.999999E+09,8.999999E+09,8.999999E+09]];
	LOCAL CONST Robtarget Tr_meulage_bavure_P28 :=[[110.9894296875,14.817318359375,95.5169140625],[0.576385001734185,-0.569893800428433,-0.411774684713817,0.416464878516733],[0,0,0,0],[8.999999E+09,8.999999E+09,8.999999E+09,8.999999E+09,8.999999E+09,8.999999E+09]];
	LOCAL CONST Robtarget Tr_meulage_bavure_P29 :=[[110.26734375,12.4955107421875,95.8813515625],[0.576462964602485,-0.57022802753016,-0.411585747558419,0.416086072186459],[0,0,0,0],[8.999999E+09,8.999999E+09,8.999999E+09,8.999999E+09,8.999999E+09,8.999999E+09]];
	LOCAL CONST Robtarget Tr_meulage_bavure_P30 :=[[109.3398046875,9.745515625,96.315140625],[0.576468070992839,-0.570475815963387,-0.411500844829266,0.415823233155031],[0,0,0,0],[8.999999E+09,8.999999E+09,8.999999E+09,8.999999E+09,8.999999E+09,8.999999E+09]];
	LOCAL CONST Robtarget Tr_meulage_bavure_P31 :=[[107.5775859375,4.87170166015625,97.0874609375],[0.576384882201262,-0.570627827770445,-0.41153959263507,0.415691608572487],[0,0,0,0],[8.999999E+09,8.999999E+09,8.999999E+09,8.999999E+09,8.999999E+09,8.999999E+09]];
	LOCAL CONST Robtarget Tr_meulage_bavure_P32 :=[[106.7702265625,2.53833129882813,97.456140625],[0.576194531069146,-0.570668712944557,-0.41172700966355,0.415713786090529],[0,0,0,0],[8.999999E+09,8.999999E+09,8.999999E+09,8.999999E+09,8.999999E+09,8.999999E+09]];
	LOCAL CONST Robtarget Tr_meulage_bavure_P33 :=[[104.9886640625,-2.732484375,98.2876875],[0.575881420174394,-0.570570583491102,-0.412088458738798,0.415924153334269],[0,0,0,0],[8.999999E+09,8.999999E+09,8.999999E+09,8.999999E+09,8.999999E+09,8.999999E+09]];
	LOCAL CONST Robtarget Tr_meulage_bavure_P34 :=[[104.60746875,-4.03763671875,98.4918125],[0.5754380561577,-0.570331276218252,-0.412632098638737,0.416326830826095],[0,0,0,0],[8.999999E+09,8.999999E+09,8.999999E+09,8.999999E+09,8.999999E+09,8.999999E+09]];
	LOCAL CONST Robtarget Tr_meulage_bavure_P35 :=[[103.801203125,-6.7024951171875,98.9094296875],[0.574873650922935,-0.569960034133665,-0.413344465007026,0.416907901355854],[0,0,0,0],[8.999999E+09,8.999999E+09,8.999999E+09,8.999999E+09,8.999999E+09,8.999999E+09]];
	LOCAL CONST Robtarget Tr_meulage_bavure_P36 :=[[102.8564375,-9.4344658203125,99.3410625],[0.574222510145913,-0.569489395448512,-0.414178124906992,0.417620423545047],[0,0,0,0],[8.999999E+09,8.999999E+09,8.999999E+09,8.999999E+09,8.999999E+09,8.999999E+09]];
	LOCAL CONST Robtarget Tr_meulage_bavure_P37 :=[[102.1071328125,-11.822208984375,99.7160546875],[0.573536775747134,-0.568962567143311,-0.415063820855947,0.418400751280083],[0,0,0,0],[8.999999E+09,8.999999E+09,8.999999E+09,8.999999E+09,8.999999E+09,8.999999E+09]];
	LOCAL CONST Robtarget Tr_meulage_bavure_P38 :=[[101.4886171875,-13.6009853515625,99.9971953125],[0.572871147429475,-0.568438536478559,-0.415925348453687,0.419168681085109],[0,0,0,0],[8.999999E+09,8.999999E+09,8.999999E+09,8.999999E+09,8.999999E+09,8.999999E+09]];
	LOCAL CONST Robtarget Tr_meulage_bavure_P39 :=[[100.8492890625,-15.5669404296875,100.3066015625],[0.572284142024175,-0.567977544045324,-0.416682988352525,0.419842419802366],[0,0,0,0],[8.999999E+09,8.999999E+09,8.999999E+09,8.999999E+09,8.999999E+09,8.999999E+09]];
	LOCAL CONST Robtarget Tr_meulage_bavure_P40 :=[[99.7165625,-19.96378125,100.9897734375],[0.571837284431263,-0.567629547935566,-0.417257741312327,0.420350798452529],[0,0,0,0],[8.999999E+09,8.999999E+09,8.999999E+09,8.999999E+09,8.999999E+09,8.999999E+09]];
	LOCAL CONST Robtarget Tr_meulage_bavure_P41 :=[[98.7682890625,-23.97071484375,101.609875],[0.571558136925635,-0.567435541032057,-0.417609203592722,0.420643264491904],[0,0,0,0],[8.999999E+09,8.999999E+09,8.999999E+09,8.999999E+09,8.999999E+09,8.999999E+09]];
	LOCAL CONST Robtarget Tr_meulage_bavure_P42 :=[[98.39775,-25.11787890625,101.79034375],[0.571463464418966,-0.567399931520206,-0.417719167816813,0.420710735997512],[0,0,0,0],[8.999999E+09,8.999999E+09,8.999999E+09,8.999999E+09,8.999999E+09,8.999999E+09]];
	LOCAL CONST Robtarget Tr_meulage_bavure_P43 :=[[98.2493359375,-25.80449609375,101.8961796875],[0.571538785080823,-0.567512048942939,-0.417606214531194,0.420569305867475],[0,0,0,0],[8.999999E+09,8.999999E+09,8.999999E+09,8.999999E+09,8.999999E+09,8.999999E+09]];
	LOCAL CONST Robtarget Tr_meulage_bavure_P44 :=[[97.184359375,-29.44232421875,102.4652109375],[0.571754644850088,-0.567741186250557,-0.417310260756414,0.420260297666307],[0,0,0,0],[8.999999E+09,8.999999E+09,8.999999E+09,8.999999E+09,8.999999E+09,8.999999E+09]];
	LOCAL CONST Robtarget Tr_meulage_bavure_P45 :=[[96.388296875,-32.202794921875,102.8966484375],[0.572057526429172,-0.568042480277886,-0.41690061514159,0.419847358155377],[0,0,0,0],[8.999999E+09,8.999999E+09,8.999999E+09,8.999999E+09,8.999999E+09,8.999999E+09]];
	LOCAL CONST Robtarget Tr_meulage_bavure_P46 :=[[95.5962734375,-34.6359140625,103.279609375],[0.572392062390525,-0.568359802574085,-0.416452206424641,0.419406749462042],[0,0,0,0],[8.999999E+09,8.999999E+09,8.999999E+09,8.999999E+09,8.999999E+09,8.999999E+09]];
	LOCAL CONST Robtarget Tr_meulage_bavure_P47 :=[[94.9805703125,-36.83403125,103.6226171875],[0.572703468136932,-0.568633041533756,-0.416041032726652,0.419019165131789],[0,0,0,0],[8.999999E+09,8.999999E+09,8.999999E+09,8.999999E+09,8.999999E+09,8.999999E+09]];
	LOCAL CONST Robtarget Tr_meulage_bavure_P48 :=[[94.24815625,-38.9423046875,103.9558125],[0.572936974506232,-0.568811202335942,-0.415740671855235,0.41875617381257],[0,0,0,0],[8.999999E+09,8.999999E+09,8.999999E+09,8.999999E+09,8.999999E+09,8.999999E+09]];
	LOCAL CONST Robtarget Tr_meulage_bavure_P49 :=[[93.68078125,-40.8864921875,104.2598671875],[0.573070764187614,-0.568870830728034,-0.415581688175399,0.418649898642656],[0,0,0,0],[8.999999E+09,8.999999E+09,8.999999E+09,8.999999E+09,8.999999E+09,8.999999E+09]];
	LOCAL CONST Robtarget Tr_meulage_bavure_P50 :=[[93.05490625,-42.77521875,104.55746875],[0.573097887376343,-0.56880901393006,-0.415572462410322,0.418705917850353],[0,0,0,0],[8.999999E+09,8.999999E+09,8.999999E+09,8.999999E+09,8.999999E+09,8.999999E+09]];
	LOCAL CONST Robtarget Tr_meulage_bavure_P51 :=[[92.552609375,-44.53103515625,104.831765625],[0.57303652488162,-0.568645442611728,-0.415687701995748,0.418897644011043],[0,0,0,0],[8.999999E+09,8.999999E+09,8.999999E+09,8.999999E+09,8.999999E+09,8.999999E+09]];
	LOCAL CONST Robtarget Tr_meulage_bavure_P52 :=[[91.432859375,-48.5715859375,105.461921875],[0.572916657911935,-0.568413020121276,-0.415885492693601,0.419180627666199],[0,0,0,0],[8.999999E+09,8.999999E+09,8.999999E+09,8.999999E+09,8.999999E+09,8.999999E+09]];
	LOCAL CONST Robtarget Tr_meulage_bavure_P53 :=[[91.2320390625,-49.15887890625,105.554640625],[0.572777306783679,-0.568147856495335,-0.416113508089247,0.419504133923674],[0,0,0,0],[8.999999E+09,8.999999E+09,8.999999E+09,8.999999E+09,8.999999E+09,8.999999E+09]];
	LOCAL CONST Robtarget Tr_meulage_bavure_P54 :=[[91.142140625,-49.2201640625,105.5663671875],[0.572638744427516,-0.567873206106166,-0.416343217077854,0.419837130040262],[0,0,0,0],[8.999999E+09,8.999999E+09,8.999999E+09,8.999999E+09,8.999999E+09,8.999999E+09]];
	LOCAL CONST Robtarget Tr_meulage_bavure_P55 :=[[91.0502890625,-49.76480859375,105.6495546875],[0.572509516598146,-0.567595585812614,-0.416563635951528,0.420170015081318],[0,0,0,0],[8.999999E+09,8.999999E+09,8.999999E+09,8.999999E+09,8.999999E+09,8.999999E+09]];
	LOCAL CONST Robtarget Tr_meulage_bavure_P56 :=[[88.28159375,-59.0003671875,107.0961171875],[0.572357639991232,-0.567300827599266,-0.416812582223046,0.420527970828828],[0,0,0,0],[8.999999E+09,8.999999E+09,8.999999E+09,8.999999E+09,8.999999E+09,8.999999E+09]];
	LOCAL CONST Robtarget Tr_meulage_bavure_P57 :=[[87.94409375,-60.14712890625,107.275546875],[0.572147378037578,-0.566948435763177,-0.417139629603424,0.420964818488113],[0,0,0,0],[8.999999E+09,8.999999E+09,8.999999E+09,8.999999E+09,8.999999E+09,8.999999E+09]];
	LOCAL CONST Robtarget Tr_meulage_bavure_P58 :=[[87.2657109375,-62.4107890625,107.63009375],[0.57184389008616,-0.566504903772261,-0.41759092729008,0.421526484124212],[0,0,0,0],[8.999999E+09,8.999999E+09,8.999999E+09,8.999999E+09,8.999999E+09,8.999999E+09]];
	LOCAL CONST Robtarget Tr_meulage_bavure_P59 :=[[86.87921875,-63.60864453125,107.81853125],[0.571418383201938,-0.565947723898588,-0.418202520445892,0.422245020154879],[0,0,0,0],[8.999999E+09,8.999999E+09,8.999999E+09,8.999999E+09,8.999999E+09,8.999999E+09]];
	LOCAL CONST Robtarget Tr_meulage_bavure_P60 :=[[86.130140625,-66.125328125,108.2125546875],[0.570869857035179,-0.56529231118974,-0.418969701199886,0.423103531910186],[0,0,0,0],[8.999999E+09,8.999999E+09,8.999999E+09,8.999999E+09,8.999999E+09,8.999999E+09]];
	LOCAL CONST Robtarget Tr_meulage_bavure_P61 :=[[84.367140625,-71.6382109375,109.0793125],[0.570247329580982,-0.564564210214913,-0.41983257730619,0.424058772674982],[0,0,0,0],[8.999999E+09,8.999999E+09,8.999999E+09,8.999999E+09,8.999999E+09,8.999999E+09]];
	LOCAL CONST Robtarget Tr_meulage_bavure_P62 :=[[83.5265703125,-74.4086015625,109.51353125],[0.569602077039325,-0.563849902301193,-0.420711898284035,0.425003835452888],[0,0,0,0],[8.999999E+09,8.999999E+09,8.999999E+09,8.999999E+09,8.999999E+09,8.999999E+09]];
	LOCAL CONST Robtarget Tr_meulage_bavure_P63 :=[[82.4703515625,-77.9844765625,110.07315625],[0.569030746578373,-0.563228696556322,-0.42148458866843,0.425826474445788],[0,0,0,0],[8.999999E+09,8.999999E+09,8.999999E+09,8.999999E+09,8.999999E+09,8.999999E+09]];
	LOCAL CONST Robtarget Tr_meulage_bavure_P64 :=[[82.144453125,-79.198296875,110.2621484375],[0.568609228962068,-0.562800176730382,-0.422044720508578,0.426400937736128],[0,0,0,0],[8.999999E+09,8.999999E+09,8.999999E+09,8.999999E+09,8.999999E+09,8.999999E+09]];
	LOCAL CONST Robtarget Tr_meulage_bavure_P65 :=[[81.7110390625,-80.4205546875,110.455578125],[0.568399113074227,-0.56261314972617,-0.422316041379343,0.426659176867568],[0,0,0,0],[8.999999E+09,8.999999E+09,8.999999E+09,8.999999E+09,8.999999E+09,8.999999E+09]];
	LOCAL CONST Robtarget Tr_meulage_bavure_P66 :=[[80.0921953125,-85.965859375,111.32284375],[0.568404832970286,-0.562702137028489,-0.422285138856395,0.426564780942623],[0,0,0,0],[8.999999E+09,8.999999E+09,8.999999E+09,8.999999E+09,8.999999E+09,8.999999E+09]];
	LOCAL CONST Robtarget Tr_meulage_bavure_P67 :=[[79.715703125,-87.3992890625,111.54578125],[0.568611792338657,-0.56303748252507,-0.421975218080293,0.426152951663298],[0,0,0,0],[8.999999E+09,8.999999E+09,8.999999E+09,8.999999E+09,8.999999E+09,8.999999E+09]];
	LOCAL CONST Robtarget Tr_meulage_bavure_P68 :=[[79.3652421875,-88.777390625,111.7597734375],[0.568950957899756,-0.563571924282043,-0.421470272629886,0.425493011640938],[0,0,0,0],[8.999999E+09,8.999999E+09,8.999999E+09,8.999999E+09,8.999999E+09,8.999999E+09]];
	LOCAL CONST Robtarget Tr_meulage_bavure_P69 :=[[79.0728671875,-89.6640625,111.8994375],[0.56933414600044,-0.564227498391955,-0.420882956977512,0.424692237723004],[0,0,0,0],[8.999999E+09,8.999999E+09,8.999999E+09,8.999999E+09,8.999999E+09,8.999999E+09]];
	LOCAL CONST Robtarget Tr_meulage_bavure_P70 :=[[77.702921875,-93.7926796875,112.55003125],[0.569673051566589,-0.564926214142086,-0.420326935901144,0.423858766394959],[0,0,0,0],[8.999999E+09,8.999999E+09,8.999999E+09,8.999999E+09,8.999999E+09,8.999999E+09]];
	LOCAL CONST Robtarget Tr_meulage_bavure_P71 :=[[77.2132734375,-95.1008671875,112.7578203125],[0.569895894806751,-0.56559930652863,-0.419897117412342,0.423086875624323],[0,0,0,0],[8.999999E+09,8.999999E+09,8.999999E+09,8.999999E+09,8.999999E+09,8.999999E+09]];
	LOCAL CONST Robtarget Tr_meulage_bavure_P72 :=[[76.152765625,-98.075625,113.228765625],[0.569954282599779,-0.566213660243025,-0.419654395897246,0.422426792124369],[0,0,0,0],[8.999999E+09,8.999999E+09,8.999999E+09,8.999999E+09,8.999999E+09,8.999999E+09]];
	LOCAL CONST Robtarget Tr_meulage_bavure_P73 :=[[75.737984375,-99.4916328125,113.450265625],[0.569847162223286,-0.56678093395806,-0.419597115659941,0.421867094163026],[0,0,0,0],[8.999999E+09,8.999999E+09,8.999999E+09,8.999999E+09,8.999999E+09,8.999999E+09]];
	LOCAL CONST Robtarget Tr_meulage_bavure_P74 :=[[75.4139140625,-101.2054765625,113.7130703125],[0.569601479086553,-0.567321537888819,-0.419691457629102,0.421378105818322],[0,0,0,0],[8.999999E+09,8.999999E+09,8.999999E+09,8.999999E+09,8.999999E+09,8.999999E+09]];
	LOCAL CONST Robtarget Tr_meulage_bavure_P75 :=[[74.8880546875,-102.807859375,113.96540625],[0.569258773738628,-0.567888780491345,-0.41987804394381,0.420890971306783],[0,0,0,0],[8.999999E+09,8.999999E+09,8.999999E+09,8.999999E+09,8.999999E+09,8.999999E+09]];
	LOCAL CONST Robtarget Tr_meulage_bavure_P76 :=[[73.539953125,-107.676078125,114.724609375],[0.568860983129904,-0.568540372826985,-0.42009518544275,0.420332084792553],[0,0,0,0],[8.999999E+09,8.999999E+09,8.999999E+09,8.999999E+09,8.999999E+09,8.999999E+09]];
	LOCAL CONST Robtarget Tr_meulage_bavure_P77 :=[[73.1556484375,-109.2884140625,114.974203125],[0.568453059595829,-0.56931604174537,-0.420282917049862,0.419645842685931],[0,0,0,0],[8.999999E+09,8.999999E+09,8.999999E+09,8.999999E+09,8.999999E+09,8.999999E+09]];
	LOCAL CONST Robtarget Tr_meulage_bavure_P78 :=[[72.54409375,-111.3528125,115.2973359375],[0.568047517227878,-0.570237997783662,-0.420420012668799,0.418805034595445],[0,0,0,0],[8.999999E+09,8.999999E+09,8.999999E+09,8.999999E+09,8.999999E+09,8.999999E+09]];
	LOCAL CONST Robtarget Tr_meulage_bavure_P79 :=[[71.464828125,-115.1288359375,115.887203125],[0.567638665728061,-0.571309115655891,-0.420509843329291,0.417808222994863],[0,0,0,0],[8.999999E+09,8.999999E+09,8.999999E+09,8.999999E+09,8.999999E+09,8.999999E+09]];
	LOCAL CONST Robtarget Tr_meulage_bavure_P80 :=[[70.6703203125,-117.5653046875,116.270734375],[0.567184512494468,-0.572486912367311,-0.420608135202737,0.416712443485711],[0,0,0,0],[8.999999E+09,8.999999E+09,8.999999E+09,8.999999E+09,8.999999E+09,8.999999E+09]];
	LOCAL CONST Robtarget Tr_meulage_bavure_P81 :=[[69.550859375,-121.230078125,116.845359375],[0.566640760349131,-0.573729297360307,-0.420773633105541,0.415574893063297],[0,0,0,0],[8.999999E+09,8.999999E+09,8.999999E+09,8.999999E+09,8.999999E+09,8.999999E+09]];
	LOCAL CONST Robtarget Tr_meulage_bavure_P82 :=[[68.8618671875,-123.084078125,117.139703125],[0.565951092736611,-0.574978899829487,-0.421083653649013,0.414472172782091],[0,0,0,0],[8.999999E+09,8.999999E+09,8.999999E+09,8.999999E+09,8.999999E+09,8.999999E+09]];
	LOCAL CONST Robtarget Tr_meulage_bavure_P83 :=[[66.925859375,-129.225453125,118.1044453125],[0.565081312414993,-0.576199996142668,-0.421586196795373,0.413451029114877],[0,0,0,0],[8.999999E+09,8.999999E+09,8.999999E+09,8.999999E+09,8.999999E+09,8.999999E+09]];
	LOCAL CONST Robtarget Tr_meulage_bavure_P84 :=[[66.5500625,-130.406328125,118.290046875],[0.564008246483587,-0.577361483602175,-0.422316735531825,0.412549378912327],[0,0,0,0],[8.999999E+09,8.999999E+09,8.999999E+09,8.999999E+09,8.999999E+09,8.999999E+09]];
	LOCAL CONST Robtarget Tr_meulage_bavure_P85 :=[[66.47440625,-130.6623203125,118.3301171875],[0.562749212642887,-0.578481327112672,-0.423251645478817,0.411741086668851],[0,0,0,0],[8.999999E+09,8.999999E+09,8.999999E+09,8.999999E+09,8.999999E+09,8.999999E+09]];
	LOCAL CONST Robtarget Tr_meulage_bavure_P86 :=[[66.437,-130.904765625,118.3670390625],[0.561388050354911,-0.5796266674497,-0.424279863165312,0.410929411228121],[0,0,0,0],[8.999999E+09,8.999999E+09,8.999999E+09,8.999999E+09,8.999999E+09,8.999999E+09]];
	LOCAL CONST Robtarget Tr_meulage_bavure_P87 :=[[65.51324609375,-134.12115625,118.869625],[0.560079410990633,-0.580968730331186,-0.425178001697286,0.409890295852998],[0,0,0,0],[8.999999E+09,8.999999E+09,8.999999E+09,8.999999E+09,8.999999E+09,8.999999E+09]];
	LOCAL CONST Robtarget Tr_meulage_bavure_P88 :=[[64.3776875,-137.38475,119.3854609375],[0.559086404059777,-0.582752454792378,-0.425578357263857,0.408295274351248],[0,0,0,0],[8.999999E+09,8.999999E+09,8.999999E+09,8.999999E+09,8.999999E+09,8.999999E+09]];
	LOCAL CONST Robtarget Tr_meulage_bavure_P89 :=[[61.7365234375,-146.514921875,120.812671875],[0.558769547865397,-0.585361240210725,-0.424948819968993,0.405644316173938],[0,0,0,0],[8.999999E+09,8.999999E+09,8.999999E+09,8.999999E+09,8.999999E+09,8.999999E+09]];
	LOCAL CONST Robtarget Tr_meulage_bavure_P90 :=[[61.22276171875,-148.260125,121.0857421875],[0.559593950719884,-0.589284703020883,-0.422574886970513,0.401283707624866],[0,0,0,0],[8.999999E+09,8.999999E+09,8.999999E+09,8.999999E+09,8.999999E+09,8.999999E+09]];
	LOCAL CONST Robtarget Tr_meulage_bavure_P91 :=[[60.7982421875,-150.0098125,121.356828125],[0.562139357106955,-0.595139271358024,-0.417493927182532,0.39434428060329],[0,0,0,0],[8.999999E+09,8.999999E+09,8.999999E+09,8.999999E+09,8.999999E+09,8.999999E+09]];
	LOCAL CONST Robtarget Tr_meulage_bavure_P92 :=[[60.07436328125,-152.97953125,121.81703125],[0.567048742232414,-0.603633313042138,-0.408469068554058,0.383712870976449],[0,0,0,0],[8.999999E+09,8.999999E+09,8.999999E+09,8.999999E+09,8.999999E+09,8.999999E+09]];
	LOCAL CONST Robtarget Tr_meulage_bavure_P93 :=[[59.62365234375,-154.5715625,122.0656015625],[0.574947364243679,-0.615456450890923,-0.393959004430782,0.368028787235322],[0,0,0,0],[8.999999E+09,8.999999E+09,8.999999E+09,8.999999E+09,8.999999E+09,8.999999E+09]];
	LOCAL CONST Robtarget Tr_meulage_bavure_P94 :=[[58.90265234375,-156.590140625,122.3852109375],[0.58630498344365,-0.631166357867292,-0.37205786837186,0.345613132951089],[0,0,0,0],[8.999999E+09,8.999999E+09,8.999999E+09,8.999999E+09,8.999999E+09,8.999999E+09]];
	LOCAL CONST Robtarget Tr_meulage_bavure_P95 :=[[58.402796875,-157.916796875,122.5960390625],[0.601163515094423,-0.650840242739021,-0.340620594275455,0.314622022919829],[0,0,0,0],[8.999999E+09,8.999999E+09,8.999999E+09,8.999999E+09,8.999999E+09,8.999999E+09]];
	LOCAL CONST Robtarget Tr_meulage_bavure_P96 :=[[56.97616796875,-159.556625,122.8806328125],[0.618658741492182,-0.673600897074773,-0.297827903502894,0.273535615469797],[0,0,0,0],[8.999999E+09,8.999999E+09,8.999999E+09,8.999999E+09,8.999999E+09,8.999999E+09]];
	LOCAL CONST Robtarget Tr_meulage_bavure_P97 :=[[56.5917265625,-159.968640625,122.9529140625],[0.636627268751023,-0.697114849390011,-0.243494518501396,0.222366874561675],[0,0,0,0],[8.999999E+09,8.999999E+09,8.999999E+09,8.999999E+09,8.999999E+09,8.999999E+09]];
	LOCAL CONST Robtarget Tr_meulage_bavure_P98 :=[[55.653109375,-160.169046875,123.010375],[0.651910892057291,-0.717876530363823,-0.180829848802963,0.164213403081976],[0,0,0,0],[8.999999E+09,8.999999E+09,8.999999E+09,8.999999E+09,8.999999E+09,8.999999E+09]];
	LOCAL CONST Robtarget Tr_meulage_bavure_P99 :=[[50.71801953125,-160.75971875,123.244109375],[0.661900353063132,-0.732941848317731,-0.116602038543167,0.105300209909894],[0,0,0,0],[8.999999E+09,8.999999E+09,8.999999E+09,8.999999E+09,8.999999E+09,8.999999E+09]];
	LOCAL CONST Robtarget Tr_meulage_bavure_P100 :=[[50.3380078125,-160.6849375,123.2443359375],[0.666165125897887,-0.741693780992938,-0.0581744039348707,0.0522503492875811],[0,0,0,0],[8.999999E+09,8.999999E+09,8.999999E+09,8.999999E+09,8.999999E+09,8.999999E+09]];
	LOCAL CONST Robtarget Tr_meulage_bavure_P101 :=[[39.9571875,-157.701578125,123.1116953125],[0.66617483857735,-0.745674320653676,-0.0100299347598202,0.00896060114247633],[0,0,0,0],[8.999999E+09,8.999999E+09,8.999999E+09,8.999999E+09,8.999999E+09,8.999999E+09]];
	LOCAL CONST Robtarget Tr_meulage_bavure_P102 :=[[39.74321484375,-157.635015625,123.1082109375],[0.663893653347438,-0.746959757854253,0.0269114980712388,-0.0239187889089112],[0,0,0,0],[8.999999E+09,8.999999E+09,8.999999E+09,8.999999E+09,8.999999E+09,8.999999E+09]];
	LOCAL CONST Robtarget Tr_meulage_bavure_P103 :=[[39.71712890625,-157.62671875,123.1077578125],[0.660747252483121,-0.747153653835886,0.0538852709425396,-0.047653577737053],[0,0,0,0],[8.999999E+09,8.999999E+09,8.999999E+09,8.999999E+09,8.999999E+09,8.999999E+09]];
	LOCAL CONST Robtarget Tr_meulage_bavure_P104 :=[[39.6085546875,-157.596359375,123.1065],[0.657548729119434,-0.747126578994209,0.0729026529059439,-0.0641618811530865],[0,0,0,0],[8.999999E+09,8.999999E+09,8.999999E+09,8.999999E+09,8.999999E+09,8.999999E+09]];
	LOCAL CONST Robtarget Tr_meulage_bavure_P105 :=[[36.7258984375,-156.681359375,123.056875],[0.654628287837988,-0.747259531440959,0.0859769137816713,-0.0753191060058585],[0,0,0,0],[8.999999E+09,8.999999E+09,8.999999E+09,8.999999E+09,8.999999E+09,8.999999E+09]];
